Yaskawa INFORM job: DEMO_ROOF_SIDE_0625_3PAINT_22.JBI

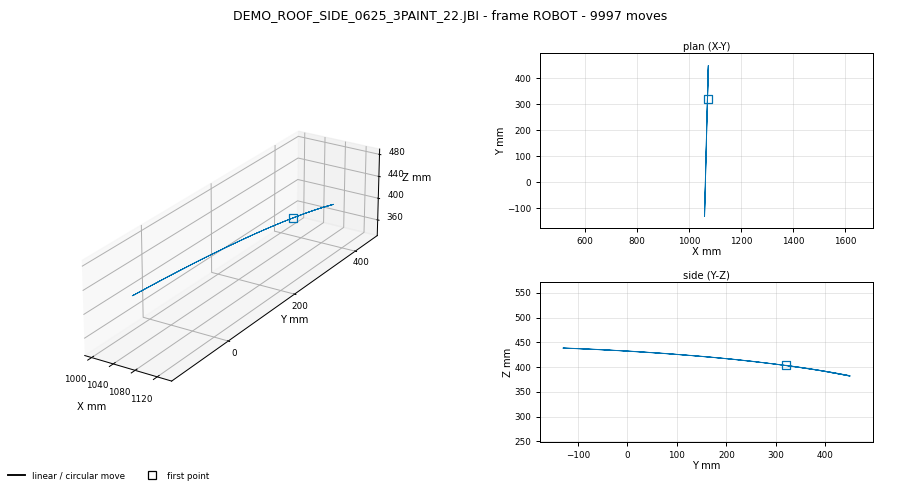
[picture p0: tool path of DEMO_ROOF_SIDE_0625_3PAINT_22.JBI in frame ROBOT, 9997 of 9997 moves have a stored position in this frame; points joined in program order, loops and branches not executed]
/JOB
//NAME DEMO_ROOF_SIDE_0625_3PAINT22
//POS
///NPOS 9997,0,0,0,0,0
///TOOL 0
///USER 0
///POSTYPE ROBOT
///RECTAN
///RCONF 1,0,0,0,0,0,0,0,0,0,0,0,0,0,0,0,0,0,0,0,0,0,0,0
C00000=1070.803,320.460,403.795,174.603,31.122,155.627
C00001=1070.809,320.707,403.762,174.607,31.127,155.628
C00002=1070.815,320.954,403.728,174.610,31.131,155.629
C00003=1070.822,321.203,403.695,174.613,31.136,155.630
C00004=1070.827,321.451,403.662,174.616,31.140,155.630
C00005=1070.834,321.698,403.629,174.620,31.145,155.631
C00006=1070.840,321.946,403.595,174.622,31.150,155.632
C00007=1070.846,322.193,403.562,174.626,31.155,155.633
C00008=1070.852,322.442,403.529,174.629,31.159,155.634
C00009=1070.859,322.689,403.495,174.633,31.164,155.635
C00010=1070.864,322.937,403.462,174.635,31.169,155.636
C00011=1070.870,323.184,403.429,174.639,31.173,155.636
C00012=1070.876,323.431,403.395,174.642,31.178,155.637
C00013=1070.883,323.680,403.362,174.645,31.183,155.638
C00014=1070.889,323.928,403.329,174.648,31.187,155.639
C00015=1070.895,324.175,403.295,174.652,31.192,155.640
C00016=1070.901,324.423,403.262,174.654,31.197,155.641
C00017=1070.908,324.670,403.228,174.658,31.201,155.642
C00018=1070.914,324.918,403.195,174.661,31.206,155.643
C00019=1070.920,325.165,403.161,174.665,31.211,155.643
C00020=1070.926,325.414,403.127,174.667,31.215,155.644
C00021=1070.933,325.661,403.094,174.671,31.220,155.645
C00022=1070.939,325.909,403.061,174.674,31.225,155.646
C00023=1070.946,326.156,403.027,174.677,31.230,155.647
C00024=1070.951,326.404,402.994,174.680,31.234,155.648
C00025=1070.957,326.651,402.959,174.684,31.239,155.649
C00026=1070.964,326.900,402.926,174.687,31.244,155.650
C00027=1070.970,327.147,402.892,174.690,31.249,155.650
C00028=1070.977,327.395,402.858,174.693,31.253,155.651
C00029=1070.983,327.643,402.825,174.697,31.258,155.652
C00030=1070.989,327.890,402.792,174.700,31.263,155.653
C00031=1070.996,328.138,402.757,174.703,31.268,155.654
C00032=1071.001,328.385,402.724,174.707,31.273,155.655
C00033=1071.008,328.633,402.690,174.710,31.277,155.656
C00034=1071.014,328.880,402.656,174.713,31.282,155.657
C00035=1071.022,329.128,402.622,174.716,31.287,155.658
C00036=1071.027,329.376,402.589,174.720,31.292,155.658
C00037=1071.034,329.624,402.554,174.722,31.296,155.659
C00038=1071.040,329.871,402.521,174.726,31.301,155.660
C00039=1071.047,330.119,402.487,174.730,31.306,155.661
C00040=1071.052,330.366,402.453,174.733,31.311,155.662
C00041=1071.058,330.589,402.423,174.735,31.315,155.663
C00042=1071.064,330.812,402.392,174.739,31.319,155.664
C00043=1071.070,331.035,402.362,174.742,31.324,155.664
C00044=1071.075,331.258,402.331,174.745,31.328,155.665
C00045=1071.081,331.480,402.300,174.747,31.332,155.666
C00046=1071.086,331.703,402.270,174.751,31.337,155.667
C00047=1071.092,331.926,402.239,174.754,31.341,155.668
C00048=1071.098,332.149,402.208,174.757,31.345,155.668
C00049=1071.104,332.397,402.174,174.760,31.350,155.669
C00050=1071.110,332.645,402.140,174.763,31.355,155.670
C00051=1071.116,332.892,402.105,174.767,31.360,155.671
C00052=1071.122,333.139,402.071,174.770,31.365,155.672
C00053=1071.129,333.387,402.036,174.773,31.370,155.673
C00054=1071.135,333.635,402.002,174.777,31.375,155.674
C00055=1071.141,333.882,401.968,174.780,31.380,155.675
C00056=1071.147,334.130,401.933,174.783,31.385,155.676
C00057=1071.153,334.377,401.899,174.787,31.390,155.677
C00058=1071.160,334.625,401.865,174.790,31.395,155.678
C00059=1071.166,334.872,401.831,174.794,31.400,155.679
C00060=1071.172,335.120,401.796,174.797,31.405,155.680
C00061=1071.178,335.367,401.762,174.800,31.410,155.681
C00062=1071.185,335.615,401.727,174.804,31.415,155.682
C00063=1071.191,335.863,401.693,174.806,31.420,155.683
C00064=1071.197,336.110,401.658,174.810,31.425,155.684
C00065=1071.204,336.358,401.624,174.814,31.430,155.684
C00066=1071.210,336.605,401.590,174.817,31.435,155.685
C00067=1071.216,336.853,401.555,174.820,31.440,155.686
C00068=1071.223,337.100,401.520,174.824,31.445,155.687
C00069=1071.229,337.348,401.486,174.827,31.450,155.688
C00070=1071.235,337.596,401.452,174.831,31.455,155.689
C00071=1071.242,337.843,401.416,174.834,31.460,155.690
C00072=1071.248,338.090,401.382,174.837,31.465,155.691
C00073=1071.255,338.338,401.347,174.841,31.470,155.692
C00074=1071.260,338.586,401.312,174.844,31.476,155.693
C00075=1071.266,338.833,401.277,174.847,31.480,155.694
C00076=1071.273,339.081,401.243,174.851,31.486,155.695
C00077=1071.280,339.328,401.208,174.855,31.491,155.696
C00078=1071.285,339.575,401.173,174.858,31.496,155.697
C00079=1071.292,339.823,401.138,174.861,31.501,155.698
C00080=1071.298,340.071,401.104,174.865,31.506,155.699
C00081=1071.304,340.317,401.069,174.869,31.511,155.700
C00082=1071.310,340.565,401.033,174.871,31.517,155.701
C00083=1071.317,340.813,400.999,174.875,31.522,155.702
C00084=1071.323,341.060,400.964,174.879,31.527,155.703
C00085=1071.329,341.307,400.928,174.883,31.532,155.704
C00086=1071.335,341.555,400.894,174.885,31.537,155.705
C00087=1071.342,341.803,400.859,174.889,31.543,155.706
C00088=1071.349,342.050,400.824,174.893,31.548,155.707
C00089=1071.354,342.298,400.789,174.896,31.553,155.708
C00090=1071.361,342.545,400.754,174.899,31.558,155.709
C00091=1071.368,342.793,400.719,174.903,31.563,155.710
C00092=1071.374,343.040,400.683,174.907,31.569,155.711
C00093=1071.380,343.288,400.649,174.910,31.573,155.712
C00094=1071.386,343.535,400.614,174.913,31.579,155.713
C00095=1071.392,343.783,400.578,174.917,31.584,155.714
C00096=1071.399,344.030,400.543,174.921,31.589,155.715
C00097=1071.405,344.250,400.511,174.924,31.594,155.716
C00098=1071.410,344.470,400.480,174.926,31.599,155.717
C00099=1071.416,344.691,400.449,174.930,31.604,155.718
C00100=1071.422,344.911,400.417,174.933,31.608,155.719
C00101=1071.426,345.131,400.386,174.936,31.613,155.719
C00102=1071.432,345.352,400.354,174.939,31.617,155.720
C00103=1071.438,345.572,400.323,174.942,31.622,155.721
C00104=1071.444,345.792,400.291,174.946,31.627,155.722
C00105=1071.450,346.039,400.256,174.949,31.632,155.723
C00106=1071.456,346.287,400.221,174.953,31.638,155.724
C00107=1071.462,346.535,400.185,174.956,31.643,155.725
C00108=1071.469,346.782,400.150,174.960,31.649,155.726
C00109=1071.475,347.029,400.113,174.963,31.654,155.727
C00110=1071.482,347.276,400.078,174.967,31.659,155.728
C00111=1071.488,347.524,400.042,174.970,31.665,155.729
C00112=1071.494,347.771,400.008,174.974,31.670,155.730
C00113=1071.500,348.018,399.972,174.978,31.676,155.732
C00114=1071.507,348.266,399.936,174.982,31.681,155.733
C00115=1071.514,348.513,399.900,174.984,31.686,155.734
C00116=1071.520,348.760,399.865,174.988,31.692,155.735
C00117=1071.526,349.008,399.829,174.992,31.697,155.736
C00118=1071.532,349.256,399.794,174.996,31.703,155.737
C00119=1071.539,349.503,399.757,174.999,31.708,155.738
C00120=1071.545,349.750,399.722,175.002,31.714,155.739
C00121=1071.552,349.998,399.686,175.006,31.719,155.740
C00122=1071.558,350.245,399.650,175.010,31.725,155.741
C00123=1071.564,350.492,399.614,175.013,31.730,155.742
C00124=1071.571,350.739,399.578,175.017,31.735,155.743
C00125=1071.577,350.987,399.543,175.021,31.741,155.744
C00126=1071.583,351.234,399.507,175.025,31.747,155.745
C00127=1071.590,351.481,399.471,175.028,31.752,155.746
C00128=1071.596,351.729,399.435,175.031,31.757,155.747
C00129=1071.602,351.976,399.399,175.035,31.763,155.749
C00130=1071.609,352.223,399.364,175.039,31.769,155.750
C00131=1071.616,352.471,399.327,175.043,31.774,155.751
C00132=1071.622,352.719,399.291,175.046,31.780,155.752
C00133=1071.629,352.966,399.255,175.050,31.785,155.753
C00134=1071.635,353.213,399.218,175.054,31.791,155.754
C00135=1071.641,353.460,399.183,175.057,31.797,155.755
C00136=1071.647,353.708,399.146,175.060,31.802,155.756
C00137=1071.654,353.954,399.110,175.064,31.808,155.757
C00138=1071.660,354.202,399.075,175.068,31.813,155.758
C00139=1071.667,354.449,399.038,175.072,31.819,155.760
C00140=1071.673,354.696,399.002,175.076,31.825,155.761
C00141=1071.679,354.944,398.966,175.079,31.831,155.762
C00142=1071.686,355.191,398.929,175.083,31.837,155.763
C00143=1071.692,355.439,398.893,175.087,31.842,155.764
C00144=1071.699,355.686,398.856,175.091,31.848,155.765
C00145=1071.705,355.933,398.820,175.094,31.854,155.766
C00146=1071.711,356.180,398.783,175.097,31.859,155.767
C00147=1071.717,356.427,398.748,175.101,31.865,155.769
C00148=1071.724,356.675,398.711,175.105,31.870,155.770
C00149=1071.731,356.922,398.674,175.109,31.876,155.771
C00150=1071.737,357.169,398.638,175.112,31.882,155.772
C00151=1071.743,357.416,398.601,175.116,31.888,155.773
C00152=1071.750,357.663,398.565,175.120,31.893,155.774
C00153=1071.756,357.886,398.532,175.124,31.899,155.775
C00154=1071.762,358.108,398.499,175.127,31.904,155.776
C00155=1071.767,358.330,398.466,175.130,31.909,155.777
C00156=1071.774,358.552,398.433,175.133,31.915,155.779
C00157=1071.780,358.774,398.401,175.137,31.919,155.779
C00158=1071.785,358.996,398.368,175.141,31.925,155.780
C00159=1071.791,359.218,398.335,175.144,31.930,155.782
C00160=1071.797,359.440,398.302,175.148,31.935,155.783
C00161=1071.803,359.688,398.265,175.151,31.941,155.784
C00162=1071.810,359.935,398.228,175.155,31.947,155.785
C00163=1071.816,360.182,398.192,175.159,31.953,155.786
C00164=1071.823,360.429,398.154,175.163,31.959,155.787
C00165=1071.830,360.676,398.118,175.167,31.965,155.788
C00166=1071.836,360.923,398.082,175.170,31.971,155.790
C00167=1071.842,361.170,398.045,175.174,31.977,155.791
C00168=1071.849,361.417,398.007,175.178,31.983,155.792
C00169=1071.855,361.665,397.971,175.182,31.988,155.793
C00170=1071.861,361.912,397.934,175.186,31.995,155.795
C00171=1071.869,362.159,397.897,175.189,32.001,155.796
C00172=1071.874,362.406,397.860,175.193,32.007,155.797
C00173=1071.881,362.654,397.823,175.197,32.012,155.798
C00174=1071.888,362.900,397.786,175.201,32.018,155.799
C00175=1071.894,363.147,397.749,175.205,32.025,155.801
C00176=1071.901,363.394,397.712,175.208,32.031,155.802
C00177=1071.907,363.642,397.675,175.212,32.037,155.803
C00178=1071.914,363.889,397.637,175.216,32.042,155.804
C00179=1071.921,364.136,397.601,175.220,32.049,155.805
C00180=1071.927,364.383,397.562,175.224,32.055,155.807
C00181=1071.933,364.631,397.526,175.228,32.061,155.808
C00182=1071.940,364.877,397.489,175.231,32.067,155.809
C00183=1071.947,365.124,397.451,175.235,32.073,155.810
C00184=1071.953,365.371,397.414,175.239,32.079,155.812
C00185=1071.959,365.619,397.376,175.243,32.086,155.813
C00186=1071.966,365.865,397.339,175.247,32.092,155.814
C00187=1071.972,366.113,397.302,175.250,32.098,155.815
C00188=1071.979,366.360,397.264,175.255,32.104,155.816
C00189=1071.985,366.607,397.226,175.259,32.110,155.818
C00190=1071.992,366.854,397.189,175.263,32.117,155.819
C00191=1071.998,367.102,397.152,175.267,32.123,155.820
C00192=1072.005,367.348,397.115,175.271,32.129,155.822
C00193=1072.011,367.596,397.076,175.274,32.135,155.823
C00194=1072.018,367.842,397.039,175.278,32.142,155.824
C00195=1072.025,368.090,397.001,175.282,32.148,155.825
C00196=1072.031,368.336,396.964,175.286,32.154,155.827
C00197=1072.038,368.583,396.926,175.290,32.160,155.828
C00198=1072.044,368.830,396.889,175.295,32.167,155.829
C00199=1072.051,369.077,396.851,175.298,32.173,155.831
C00200=1072.058,369.324,396.813,175.302,32.180,155.832
C00201=1072.064,369.571,396.775,175.306,32.186,155.833
C00202=1072.071,369.818,396.738,175.310,32.192,155.834
C00203=1072.077,370.065,396.700,175.314,32.198,155.836
C00204=1072.084,370.313,396.662,175.318,32.205,155.837
C00205=1072.090,370.559,396.625,175.322,32.211,155.838
C00206=1072.097,370.806,396.587,175.326,32.217,155.840
C00207=1072.104,371.054,396.549,175.330,32.224,155.841
C00208=1072.110,371.300,396.511,175.334,32.230,155.842
C00209=1072.117,371.531,396.476,175.338,32.237,155.844
C00210=1072.123,371.762,396.441,175.342,32.242,155.845
C00211=1072.129,371.992,396.405,175.346,32.248,155.846
C00212=1072.136,372.223,396.369,175.349,32.255,155.847
C00213=1072.141,372.453,396.334,175.353,32.260,155.848
C00214=1072.148,372.683,396.299,175.356,32.267,155.850
C00215=1072.155,372.914,396.263,175.360,32.272,155.851
C00216=1072.160,373.145,396.228,175.364,32.279,155.852
C00217=1072.167,373.392,396.189,175.369,32.285,155.854
C00218=1072.174,373.638,396.152,175.373,32.292,155.855
C00219=1072.181,373.885,396.113,175.377,32.299,155.856
C00220=1072.187,374.132,396.075,175.380,32.305,155.858
C00221=1072.193,374.378,396.036,175.384,32.312,155.859
C00222=1072.200,374.626,395.998,175.389,32.318,155.860
C00223=1072.207,374.873,395.959,175.393,32.325,155.862
C00224=1072.213,375.120,395.921,175.397,32.332,155.863
C00225=1072.219,375.366,395.883,175.401,32.338,155.865
C00226=1072.227,375.613,395.845,175.405,32.345,155.866
C00227=1072.233,375.860,395.806,175.410,32.352,155.867
C00228=1072.240,376.108,395.768,175.413,32.359,155.869
C00229=1072.247,376.355,395.729,175.417,32.365,155.870
C00230=1072.253,376.601,395.691,175.421,32.372,155.872
C00231=1072.259,376.848,395.653,175.426,32.379,155.873
C00232=1072.266,377.095,395.614,175.430,32.386,155.874
C00233=1072.273,377.342,395.575,175.434,32.392,155.876
C00234=1072.280,377.589,395.536,175.438,32.399,155.877
C00235=1072.286,377.836,395.498,175.443,32.406,155.879
C00236=1072.293,378.083,395.459,175.446,32.413,155.880
C00237=1072.299,378.329,395.421,175.450,32.420,155.881
C00238=1072.306,378.576,395.382,175.455,32.426,155.883
C00239=1072.313,378.823,395.343,175.459,32.433,155.884
C00240=1072.320,379.069,395.304,175.463,32.440,155.886
C00241=1072.327,379.316,395.266,175.468,32.447,155.887
C00242=1072.333,379.563,395.227,175.472,32.454,155.889
C00243=1072.340,379.810,395.188,175.476,32.461,155.890
C00244=1072.347,380.057,395.150,175.481,32.468,155.892
C00245=1072.354,380.304,395.110,175.485,32.475,155.893
C00246=1072.361,380.550,395.071,175.488,32.482,155.895
C00247=1072.367,380.797,395.032,175.493,32.489,155.896
C00248=1072.374,381.044,394.994,175.497,32.496,155.897
C00249=1072.381,381.291,394.955,175.501,32.503,155.899
C00250=1072.388,381.538,394.916,175.506,32.510,155.900
C00251=1072.395,381.784,394.877,175.510,32.517,155.902
C00252=1072.402,382.031,394.838,175.514,32.524,155.903
C00253=1072.408,382.278,394.799,175.519,32.531,155.905
C00254=1072.415,382.525,394.759,175.523,32.538,155.906
C00255=1072.422,382.771,394.720,175.527,32.545,155.908
C00256=1072.428,383.018,394.682,175.532,32.552,155.909
C00257=1072.435,383.264,394.642,175.536,32.560,155.911
C00258=1072.442,383.512,394.603,175.540,32.567,155.912
C00259=1072.448,383.758,394.564,175.544,32.574,155.914
C00260=1072.455,384.005,394.524,175.548,32.581,155.915
C00261=1072.462,384.252,394.485,175.553,32.589,155.917
C00262=1072.469,384.498,394.445,175.557,32.596,155.919
C00263=1072.476,384.746,394.406,175.561,32.603,155.920
C00264=1072.482,384.992,394.366,175.566,32.610,155.922
C00265=1072.490,385.237,394.327,175.570,32.618,155.923
C00266=1072.496,385.482,394.289,175.575,32.625,155.925
C00267=1072.502,385.727,394.249,175.579,32.633,155.926
C00268=1072.509,385.972,394.209,175.583,32.639,155.928
C00269=1072.516,386.217,394.171,175.588,32.647,155.929
C00270=1072.523,386.462,394.131,175.592,32.654,155.931
C00271=1072.530,386.709,394.091,175.597,32.662,155.933
C00272=1072.537,386.954,394.052,175.601,32.669,155.934
C00273=1072.544,387.200,394.013,175.606,32.676,155.936
C00274=1072.550,387.447,393.973,175.610,32.684,155.937
C00275=1072.557,387.693,393.933,175.615,32.692,155.939
C00276=1072.565,387.940,393.894,175.619,32.699,155.941
C00277=1072.571,388.187,393.854,175.624,32.706,155.942
C00278=1072.578,388.433,393.814,175.628,32.714,155.944
C00279=1072.585,388.680,393.774,175.632,32.722,155.945
C00280=1072.592,388.927,393.734,175.636,32.729,155.947
C00281=1072.599,389.173,393.694,175.641,32.736,155.948
C00282=1072.606,389.420,393.655,175.645,32.744,155.950
C00283=1072.613,389.667,393.615,175.650,32.752,155.952
C00284=1072.620,389.913,393.575,175.654,32.759,155.953
C00285=1072.627,390.160,393.535,175.659,32.767,155.955
C00286=1072.634,390.407,393.495,175.663,32.774,155.957
C00287=1072.641,390.653,393.455,175.668,32.782,155.958
C00288=1072.649,390.900,393.415,175.672,32.789,155.960
C00289=1072.655,391.146,393.375,175.677,32.797,155.962
C00290=1072.662,391.392,393.334,175.681,32.805,155.963
C00291=1072.669,391.639,393.294,175.686,32.813,155.965
C00292=1072.676,391.886,393.254,175.691,32.821,155.967
C00293=1072.683,392.133,393.214,175.695,32.828,155.968
C00294=1072.690,392.378,393.174,175.700,32.836,155.970
C00295=1072.697,392.625,393.133,175.704,32.844,155.972
C00296=1072.704,392.872,393.093,175.709,32.852,155.973
C00297=1072.711,393.118,393.053,175.713,32.860,155.975
C00298=1072.718,393.365,393.012,175.718,32.868,155.977
C00299=1072.724,393.612,392.972,175.723,32.876,155.979
C00300=1072.732,393.858,392.931,175.727,32.884,155.980
C00301=1072.739,394.104,392.891,175.732,32.892,155.982
C00302=1072.746,394.352,392.851,175.737,32.900,155.984
C00303=1072.752,394.597,392.810,175.742,32.908,155.985
C00304=1072.759,394.845,392.769,175.747,32.916,155.987
C00305=1072.766,395.091,392.728,175.751,32.924,155.989
C00306=1072.774,395.337,392.688,175.756,32.932,155.991
C00307=1072.781,395.584,392.647,175.761,32.940,155.993
C00308=1072.788,395.830,392.606,175.765,32.948,155.994
C00309=1072.795,396.077,392.566,175.770,32.956,155.996
C00310=1072.801,396.323,392.525,175.775,32.964,155.998
C00311=1072.808,396.570,392.485,175.779,32.972,156.000
C00312=1072.816,396.817,392.443,175.784,32.981,156.001
C00313=1072.822,397.063,392.402,175.789,32.989,156.003
C00314=1072.830,397.309,392.361,175.793,32.997,156.005
C00315=1072.837,397.556,392.321,175.798,33.005,156.007
C00316=1072.844,397.802,392.280,175.803,33.014,156.009
C00317=1072.851,398.049,392.239,175.807,33.022,156.010
C00318=1072.859,398.295,392.198,175.812,33.030,156.012
C00319=1072.866,398.542,392.157,175.817,33.038,156.014
C00320=1072.873,398.788,392.116,175.821,33.047,156.016
C00321=1072.879,399.048,392.072,175.827,33.056,156.018
C00322=1072.887,399.307,392.029,175.832,33.065,156.020
C00323=1072.894,399.567,391.986,175.837,33.073,156.022
C00324=1072.902,399.826,391.942,175.842,33.082,156.024
C00325=1072.909,400.072,391.902,175.847,33.091,156.026
C00326=1072.916,400.318,391.860,175.852,33.100,156.028
C00327=1072.923,400.565,391.819,175.857,33.108,156.029
C00328=1072.931,400.811,391.778,175.861,33.116,156.031
C00329=1072.938,401.058,391.735,175.866,33.125,156.033
C00330=1072.945,401.304,391.694,175.871,33.134,156.035
C00331=1072.952,401.550,391.653,175.877,33.142,156.037
C00332=1072.959,401.797,391.612,175.881,33.151,156.039
C00333=1072.966,402.043,391.571,175.886,33.160,156.041
C00334=1072.974,402.289,391.529,175.891,33.168,156.043
C00335=1072.981,402.536,391.488,175.896,33.177,156.045
C00336=1072.988,402.783,391.446,175.901,33.186,156.047
C00337=1072.995,403.029,391.404,175.906,33.195,156.049
C00338=1073.002,403.275,391.363,175.911,33.203,156.050
C00339=1073.010,403.522,391.321,175.916,33.212,156.052
C00340=1073.017,403.768,391.279,175.921,33.220,156.054
C00341=1073.024,404.015,391.238,175.926,33.229,156.056
C00342=1073.031,404.261,391.196,175.931,33.238,156.058
C00343=1073.038,404.508,391.154,175.936,33.247,156.060
C00344=1073.046,404.754,391.112,175.941,33.256,156.062
C00345=1073.053,405.000,391.070,175.946,33.265,156.064
C00346=1073.060,405.247,391.028,175.951,33.274,156.066
C00347=1073.067,405.492,390.986,175.956,33.283,156.068
C00348=1073.074,405.739,390.944,175.961,33.292,156.070
C00349=1073.082,405.985,390.902,175.966,33.301,156.072
C00350=1073.088,406.232,390.860,175.971,33.310,156.075
C00351=1073.096,406.478,390.818,175.977,33.319,156.077
C00352=1073.104,406.724,390.776,175.982,33.329,156.079
C00353=1073.111,406.971,390.734,175.987,33.337,156.081
C00354=1073.118,407.218,390.691,175.992,33.347,156.083
C00355=1073.125,407.463,390.649,175.997,33.356,156.085
C00356=1073.132,407.710,390.607,176.003,33.365,156.087
C00357=1073.140,407.956,390.565,176.008,33.374,156.089
C00358=1073.146,408.202,390.522,176.013,33.384,156.091
C00359=1073.154,408.449,390.479,176.018,33.393,156.093
C00360=1073.162,408.695,390.437,176.024,33.402,156.095
C00361=1073.168,408.941,390.395,176.029,33.412,156.097
C00362=1073.176,409.187,390.353,176.034,33.421,156.100
C00363=1073.183,409.434,390.310,176.039,33.431,156.102
C00364=1073.191,409.680,390.267,176.045,33.440,156.104
C00365=1073.198,409.926,390.225,176.050,33.449,156.106
C00366=1073.205,410.172,390.182,176.055,33.459,156.108
C00367=1073.212,410.419,390.139,176.060,33.469,156.110
C00368=1073.220,410.665,390.097,176.066,33.478,156.112
C00369=1073.227,410.911,390.054,176.071,33.488,156.115
C00370=1073.235,411.158,390.011,176.076,33.497,156.117
C00371=1073.242,411.404,389.969,176.081,33.507,156.119
C00372=1073.249,411.649,389.926,176.087,33.516,156.121
C00373=1073.257,411.896,389.883,176.092,33.526,156.123
C00374=1073.264,412.142,389.840,176.098,33.536,156.126
C00375=1073.272,412.388,389.798,176.103,33.546,156.128
C00376=1073.279,412.634,389.754,176.109,33.555,156.130
C00377=1073.287,412.898,389.709,176.114,33.566,156.132
C00378=1073.295,413.163,389.662,176.120,33.576,156.135
C00379=1073.304,413.427,389.617,176.127,33.587,156.137
C00380=1073.311,413.690,389.570,176.132,33.597,156.140
C00381=1073.319,413.936,389.527,176.137,33.607,156.142
C00382=1073.326,414.183,389.484,176.144,33.617,156.144
C00383=1073.334,414.429,389.441,176.149,33.627,156.146
C00384=1073.342,414.675,389.398,176.154,33.637,156.149
C00385=1073.350,414.921,389.354,176.160,33.647,156.151
C00386=1073.357,415.168,389.311,176.165,33.657,156.153
C00387=1073.364,415.413,389.268,176.171,33.667,156.156
C00388=1073.372,415.660,389.225,176.177,33.677,156.158
C00389=1073.379,415.905,389.181,176.182,33.687,156.160
C00390=1073.387,416.152,389.138,176.189,33.698,156.163
C00391=1073.395,416.398,389.094,176.194,33.707,156.165
C00392=1073.402,416.644,389.051,176.199,33.718,156.167
C00393=1073.410,416.890,389.007,176.205,33.728,156.170
C00394=1073.417,417.136,388.964,176.211,33.738,156.172
C00395=1073.424,417.382,388.920,176.216,33.748,156.174
C00396=1073.433,417.628,388.876,176.222,33.759,156.177
C00397=1073.439,417.874,388.832,176.228,33.770,156.179
C00398=1073.447,418.120,388.789,176.234,33.780,156.182
C00399=1073.454,418.367,388.745,176.239,33.790,156.184
C00400=1073.463,418.612,388.701,176.246,33.801,156.187
C00401=1073.470,418.858,388.657,176.251,33.811,156.189
C00402=1073.478,419.103,388.614,176.257,33.822,156.191
C00403=1073.485,419.348,388.570,176.263,33.832,156.194
C00404=1073.493,419.593,388.526,176.268,33.843,156.196
C00405=1073.501,419.839,388.482,176.275,33.853,156.199
C00406=1073.508,420.084,388.438,176.280,33.864,156.201
C00407=1073.516,420.329,388.394,176.287,33.874,156.204
C00408=1073.523,420.574,388.350,176.292,33.885,156.206
C00409=1073.531,420.820,388.306,176.299,33.896,156.209
C00410=1073.539,421.066,388.263,176.304,33.907,156.211
C00411=1073.547,421.312,388.218,176.311,33.918,156.214
C00412=1073.555,421.559,388.175,176.316,33.928,156.216
C00413=1073.562,421.805,388.130,176.323,33.939,156.219
C00414=1073.570,422.050,388.085,176.328,33.950,156.221
C00415=1073.577,422.296,388.040,176.335,33.961,156.224
C00416=1073.586,422.542,387.996,176.340,33.972,156.227
C00417=1073.594,422.788,387.952,176.347,33.983,156.229
C00418=1073.601,423.035,387.907,176.352,33.994,156.232
C00419=1073.608,423.280,387.863,176.359,34.005,156.234
C00420=1073.615,423.526,387.819,176.364,34.016,156.237
C00421=1073.623,423.771,387.774,176.371,34.028,156.240
C00422=1073.631,424.017,387.729,176.378,34.039,156.242
C00423=1073.639,424.263,387.684,176.383,34.050,156.245
C00424=1073.648,424.509,387.640,176.390,34.061,156.248
C00425=1073.655,424.755,387.595,176.395,34.073,156.250
C00426=1073.663,425.001,387.550,176.402,34.084,156.253
C00427=1073.671,425.247,387.505,176.408,34.095,156.256
C00428=1073.679,425.492,387.460,176.414,34.106,156.258
C00429=1073.686,425.738,387.415,176.421,34.118,156.261
C00430=1073.694,425.984,387.371,176.427,34.129,156.264
C00431=1073.702,426.229,387.325,176.434,34.141,156.266
C00432=1073.711,426.476,387.281,176.440,34.152,156.269
C00433=1073.719,426.757,387.229,176.447,34.166,156.272
C00434=1073.729,427.037,387.178,176.454,34.179,156.275
C00435=1073.737,427.318,387.126,176.462,34.192,156.278
C00436=1073.747,427.598,387.075,176.469,34.205,156.282
C00437=1073.755,427.844,387.029,176.475,34.217,156.284
C00438=1073.762,428.090,386.984,176.482,34.229,156.287
C00439=1073.770,428.336,386.938,176.489,34.241,156.290
C00440=1073.778,428.581,386.893,176.495,34.252,156.293
C00441=1073.786,428.828,386.848,176.501,34.264,156.296
C00442=1073.794,429.073,386.802,176.508,34.276,156.299
C00443=1073.802,429.318,386.757,176.515,34.288,156.301
C00444=1073.811,429.564,386.711,176.521,34.300,156.304
C00445=1073.818,429.810,386.666,176.528,34.313,156.307
C00446=1073.826,430.055,386.620,176.535,34.324,156.310
C00447=1073.835,430.301,386.575,176.542,34.336,156.313
C00448=1073.843,430.546,386.529,176.547,34.349,156.316
C00449=1073.850,430.792,386.483,176.554,34.361,156.319
C00450=1073.858,431.038,386.437,176.561,34.373,156.322
C00451=1073.866,431.283,386.392,176.568,34.385,156.325
C00452=1073.875,431.529,386.346,176.575,34.397,156.328
C00453=1073.883,431.774,386.300,176.581,34.410,156.331
C00454=1073.891,432.020,386.254,176.588,34.422,156.334
C00455=1073.899,432.266,386.208,176.595,34.435,156.337
C00456=1073.907,432.511,386.161,176.602,34.447,156.340
C00457=1073.915,432.757,386.116,176.609,34.460,156.343
C00458=1073.923,433.003,386.070,176.616,34.472,156.346
C00459=1073.931,433.248,386.023,176.623,34.485,156.349
C00460=1073.939,433.494,385.977,176.630,34.498,156.352
C00461=1073.947,433.738,385.931,176.636,34.510,156.355
C00462=1073.956,433.984,385.884,176.643,34.523,156.358
C00463=1073.964,434.230,385.838,176.650,34.536,156.361
C00464=1073.971,434.475,385.791,176.657,34.548,156.364
C00465=1073.980,434.721,385.745,176.665,34.561,156.368
C00466=1073.988,434.967,385.699,176.672,34.574,156.371
C00467=1073.996,435.212,385.652,176.679,34.587,156.374
C00468=1074.005,435.457,385.606,176.686,34.600,156.377
C00469=1074.013,435.703,385.559,176.693,34.613,156.380
C00470=1074.021,435.948,385.512,176.700,34.626,156.383
C00471=1074.030,436.193,385.466,176.707,34.639,156.387
C00472=1074.038,436.439,385.419,176.715,34.652,156.390
C00473=1074.047,436.684,385.372,176.722,34.665,156.393
C00474=1074.055,436.930,385.325,176.729,34.679,156.396
C00475=1074.063,437.175,385.279,176.736,34.692,156.399
C00476=1074.071,437.420,385.232,176.744,34.705,156.403
C00477=1074.080,437.666,385.185,176.751,34.718,156.406
C00478=1074.088,437.911,385.138,176.758,34.732,156.409
C00479=1074.097,438.156,385.091,176.765,34.745,156.413
C00480=1074.106,438.402,385.044,176.774,34.759,156.416
C00481=1074.114,438.647,384.996,176.781,34.772,156.419
C00482=1074.122,438.892,384.949,176.788,34.786,156.423
C00483=1074.131,439.138,384.903,176.796,34.799,156.426
C00484=1074.139,439.383,384.855,176.803,34.813,156.429
C00485=1074.147,439.629,384.808,176.810,34.827,156.433
C00486=1074.156,439.873,384.760,176.818,34.840,156.436
C00487=1074.164,440.119,384.712,176.826,34.854,156.440
C00488=1074.173,440.364,384.666,176.834,34.868,156.443
C00489=1074.186,440.768,384.587,176.846,34.891,156.449
C00490=1074.201,441.172,384.509,176.859,34.914,156.455
C00491=1074.215,441.576,384.431,176.871,34.937,156.460
C00492=1074.230,441.980,384.352,176.884,34.960,156.466
C00493=1074.238,442.225,384.304,176.892,34.975,156.470
C00494=1074.246,442.470,384.256,176.900,34.989,156.473
C00495=1074.255,442.715,384.208,176.908,35.003,156.477
C00496=1074.263,442.960,384.160,176.915,35.017,156.480
C00497=1074.272,443.205,384.112,176.924,35.032,156.484
C00498=1074.281,443.451,384.064,176.932,35.047,156.488
C00499=1074.289,443.696,384.016,176.939,35.061,156.491
C00500=1074.298,443.941,383.967,176.948,35.075,156.495
C00501=1074.307,444.186,383.920,176.955,35.090,156.499
C00502=1074.315,444.431,383.872,176.964,35.105,156.502
C00503=1074.324,444.676,383.823,176.972,35.119,156.506
C00504=1074.333,444.921,383.775,176.980,35.134,156.510
C00505=1074.342,445.166,383.726,176.988,35.149,156.514
C00506=1074.351,445.411,383.677,176.997,35.164,156.517
C00507=1074.359,445.656,383.629,177.005,35.179,156.521
C00508=1074.368,445.901,383.580,177.013,35.194,156.525
C00509=1074.377,446.146,383.532,177.021,35.209,156.529
C00510=1074.385,446.391,383.484,177.030,35.224,156.532
C00511=1074.394,446.636,383.435,177.038,35.239,156.536
C00512=1074.403,446.881,383.386,177.047,35.254,156.540
C00513=1074.412,447.126,383.338,177.054,35.269,156.544
C00514=1074.421,447.371,383.288,177.063,35.284,156.548
C00515=1074.430,447.616,383.240,177.071,35.300,156.552
C00516=1074.439,447.861,383.191,177.078,35.315,156.556
C00517=1074.448,448.105,383.142,177.085,35.330,156.560
C00518=1074.457,448.349,383.093,177.092,35.345,156.564
C00519=1074.466,448.593,383.045,177.098,35.360,156.567
C00520=1074.476,448.838,382.996,177.105,35.375,156.571
C00521=1074.487,449.082,382.948,177.111,35.389,156.575
C00522=1074.499,449.327,382.902,177.117,35.403,156.578
C00523=1074.514,449.573,382.856,177.123,35.416,156.582
C00524=1074.529,449.819,382.810,177.129,35.429,156.585
C00525=1074.173,449.816,382.569,177.111,35.579,156.625
C00526=1074.159,449.570,382.615,177.105,35.566,156.622
C00527=1074.145,449.325,382.661,177.099,35.553,156.618
C00528=1074.132,449.080,382.708,177.092,35.540,156.615
C00529=1074.120,448.835,382.755,177.087,35.526,156.611
C00530=1074.110,448.590,382.803,177.080,35.511,156.607
C00531=1074.101,448.346,382.853,177.073,35.496,156.603
C00532=1074.092,448.102,382.901,177.065,35.481,156.600
C00533=1074.083,447.858,382.950,177.059,35.466,156.596
C00534=1074.073,447.613,382.999,177.051,35.450,156.592
C00535=1074.065,447.369,383.048,177.043,35.435,156.588
C00536=1074.056,447.123,383.097,177.034,35.420,156.584
C00537=1074.047,446.878,383.146,177.027,35.405,156.580
C00538=1074.038,446.634,383.195,177.018,35.390,156.576
C00539=1074.029,446.389,383.243,177.009,35.375,156.572
C00540=1074.020,446.144,383.292,177.001,35.360,156.569
C00541=1074.011,445.899,383.341,176.992,35.345,156.565
C00542=1074.003,445.653,383.389,176.985,35.330,156.561
C00543=1073.993,445.409,383.438,176.976,35.315,156.557
C00544=1073.985,445.164,383.486,176.967,35.300,156.553
C00545=1073.976,444.919,383.536,176.959,35.285,156.550
C00546=1073.967,444.674,383.583,176.951,35.271,156.546
C00547=1073.959,444.429,383.632,176.943,35.256,156.542
C00548=1073.950,444.183,383.680,176.934,35.241,156.538
C00549=1073.941,443.939,383.728,176.927,35.227,156.535
C00550=1073.932,443.693,383.777,176.918,35.212,156.531
C00551=1073.924,443.448,383.825,176.910,35.198,156.527
C00552=1073.915,443.204,383.873,176.902,35.183,156.524
C00553=1073.907,442.958,383.921,176.894,35.169,156.520
C00554=1073.897,442.713,383.969,176.886,35.154,156.516
C00555=1073.889,442.468,384.017,176.878,35.140,156.513
C00556=1073.880,442.223,384.064,176.870,35.126,156.509
C00557=1073.872,441.978,384.112,176.862,35.112,156.506
C00558=1073.858,441.591,384.188,176.850,35.089,156.500
C00559=1073.845,441.206,384.263,176.837,35.067,156.495
C00560=1073.831,440.819,384.339,176.825,35.045,156.489
C00561=1073.817,440.433,384.413,176.813,35.023,156.484
C00562=1073.809,440.188,384.461,176.805,35.009,156.480
C00563=1073.801,439.943,384.508,176.797,34.996,156.477
C00564=1073.792,439.698,384.555,176.790,34.982,156.473
C00565=1073.784,439.453,384.603,176.783,34.968,156.470
C00566=1073.775,439.207,384.650,176.774,34.955,156.466
C00567=1073.767,438.962,384.698,176.767,34.941,156.463
C00568=1073.759,438.716,384.745,176.759,34.927,156.460
C00569=1073.750,438.472,384.792,176.752,34.914,156.456
C00570=1073.741,438.226,384.839,176.745,34.900,156.453
C00571=1073.732,437.981,384.886,176.737,34.887,156.450
C00572=1073.725,437.735,384.934,176.729,34.874,156.446
C00573=1073.716,437.490,384.980,176.722,34.860,156.443
C00574=1073.707,437.244,385.027,176.715,34.847,156.440
C00575=1073.699,436.999,385.075,176.707,34.834,156.437
C00576=1073.690,436.754,385.121,176.700,34.821,156.433
C00577=1073.682,436.508,385.168,176.693,34.808,156.430
C00578=1073.673,436.263,385.215,176.686,34.794,156.427
C00579=1073.666,436.018,385.262,176.678,34.781,156.424
C00580=1073.657,435.772,385.308,176.670,34.768,156.420
C00581=1073.649,435.527,385.355,176.663,34.755,156.417
C00582=1073.640,435.281,385.402,176.656,34.743,156.414
C00583=1073.632,435.036,385.448,176.649,34.729,156.411
C00584=1073.624,434.791,385.495,176.642,34.717,156.408
C00585=1073.615,434.545,385.541,176.635,34.704,156.405
C00586=1073.607,434.300,385.587,176.628,34.691,156.402
C00587=1073.599,434.054,385.634,176.621,34.678,156.398
C00588=1073.591,433.808,385.680,176.614,34.666,156.395
C00589=1073.583,433.563,385.726,176.606,34.653,156.392
C00590=1073.574,433.318,385.773,176.599,34.640,156.389
C00591=1073.567,433.073,385.819,176.592,34.628,156.386
C00592=1073.558,432.827,385.866,176.585,34.615,156.383
C00593=1073.550,432.581,385.912,176.578,34.602,156.380
C00594=1073.542,432.336,385.958,176.571,34.590,156.377
C00595=1073.534,432.090,386.004,176.564,34.578,156.374
C00596=1073.526,431.845,386.050,176.558,34.565,156.371
C00597=1073.517,431.599,386.096,176.552,34.553,156.368
C00598=1073.510,431.354,386.142,176.545,34.541,156.365
C00599=1073.502,431.107,386.188,176.538,34.529,156.362
C00600=1073.494,430.862,386.234,176.531,34.516,156.359
C00601=1073.485,430.617,386.280,176.524,34.504,156.356
C00602=1073.477,430.371,386.325,176.517,34.492,156.353
C00603=1073.469,430.126,386.371,176.510,34.480,156.350
C00604=1073.461,429.880,386.417,176.504,34.468,156.347
C00605=1073.453,429.634,386.463,176.497,34.455,156.344
C00606=1073.444,429.388,386.508,176.490,34.444,156.342
C00607=1073.437,429.143,386.554,176.484,34.432,156.339
C00608=1073.429,428.898,386.599,176.477,34.420,156.336
C00609=1073.421,428.651,386.645,176.471,34.408,156.333
C00610=1073.413,428.406,386.690,176.464,34.396,156.330
C00611=1073.405,428.160,386.735,176.457,34.384,156.327
C00612=1073.397,427.914,386.781,176.451,34.373,156.324
C00613=1073.389,427.669,386.826,176.444,34.361,156.322
C00614=1073.381,427.386,386.878,176.437,34.347,156.318
C00615=1073.371,427.104,386.930,176.429,34.334,156.315
C00616=1073.361,426.821,386.982,176.422,34.320,156.312
C00617=1073.352,426.539,387.033,176.414,34.307,156.309
C00618=1073.345,426.293,387.079,176.408,34.296,156.306
C00619=1073.337,426.048,387.123,176.402,34.284,156.303
C00620=1073.328,425.802,387.169,176.395,34.273,156.301
C00621=1073.320,425.556,387.214,176.388,34.262,156.298
C00622=1073.313,425.310,387.259,176.383,34.250,156.295
C00623=1073.305,425.065,387.304,176.376,34.239,156.292
C00624=1073.297,424.819,387.349,176.370,34.228,156.290
C00625=1073.289,424.573,387.393,176.364,34.216,156.287
C00626=1073.282,424.327,387.438,176.357,34.205,156.284
C00627=1073.273,424.082,387.483,176.351,34.194,156.282
C00628=1073.266,423.835,387.528,176.345,34.183,156.279
C00629=1073.257,423.589,387.573,176.338,34.171,156.277
C00630=1073.249,423.343,387.617,176.332,34.160,156.274
C00631=1073.242,423.097,387.662,176.326,34.149,156.271
C00632=1073.234,422.852,387.706,176.320,34.138,156.269
C00633=1073.227,422.606,387.751,176.314,34.127,156.266
C00634=1073.219,422.361,387.795,176.308,34.116,156.263
C00635=1073.211,422.115,387.839,176.301,34.105,156.261
C00636=1073.204,421.869,387.884,176.296,34.094,156.258
C00637=1073.196,421.622,387.928,176.289,34.083,156.256
C00638=1073.189,421.376,387.973,176.284,34.073,156.253
C00639=1073.181,421.131,388.017,176.277,34.062,156.251
C00640=1073.173,420.885,388.062,176.272,34.051,156.248
C00641=1073.165,420.639,388.105,176.265,34.040,156.246
C00642=1073.157,420.393,388.149,176.259,34.030,156.243
C00643=1073.149,420.146,388.193,176.253,34.019,156.241
C00644=1073.142,419.900,388.238,176.247,34.008,156.238
C00645=1073.134,419.655,388.281,176.241,33.998,156.236
C00646=1073.126,419.409,388.326,176.235,33.987,156.233
C00647=1073.119,419.163,388.369,176.230,33.977,156.231
C00648=1073.111,418.917,388.414,176.223,33.966,156.228
C00649=1073.103,418.670,388.457,176.218,33.956,156.226
C00650=1073.095,418.425,388.501,176.211,33.945,156.223
C00651=1073.088,418.179,388.545,176.206,33.935,156.221
C00652=1073.081,417.932,388.589,176.200,33.924,156.219
C00653=1073.073,417.686,388.633,176.194,33.914,156.216
C00654=1073.065,417.441,388.677,176.188,33.903,156.214
C00655=1073.058,417.195,388.720,176.183,33.893,156.211
C00656=1073.050,416.948,388.764,176.177,33.883,156.209
C00657=1073.043,416.703,388.807,176.171,33.872,156.207
C00658=1073.035,416.456,388.851,176.166,33.863,156.204
C00659=1073.027,416.210,388.894,176.159,33.852,156.202
C00660=1073.020,415.964,388.938,176.154,33.842,156.199
C00661=1073.012,415.718,388.981,176.148,33.832,156.197
C00662=1073.005,415.472,389.024,176.143,33.821,156.195
C00663=1072.997,415.226,389.068,176.136,33.812,156.192
C00664=1072.989,414.979,389.112,176.131,33.801,156.190
C00665=1072.982,414.734,389.155,176.126,33.792,156.188
C00666=1072.975,414.487,389.199,176.120,33.782,156.186
C00667=1072.967,414.242,389.241,176.115,33.772,156.183
C00668=1072.959,413.995,389.284,176.108,33.762,156.181
C00669=1072.951,413.749,389.328,176.103,33.752,156.179
C00670=1072.944,413.485,389.374,176.098,33.742,156.176
C00671=1072.936,413.221,389.420,176.091,33.731,156.174
C00672=1072.927,412.957,389.467,176.085,33.720,156.171
C00673=1072.919,412.692,389.512,176.080,33.710,156.169
C00674=1072.912,412.447,389.555,176.074,33.700,156.167
C00675=1072.905,412.200,389.598,176.069,33.690,156.165
C00676=1072.897,411.954,389.641,176.062,33.681,156.162
C00677=1072.889,411.708,389.683,176.057,33.671,156.160
C00678=1072.882,411.462,389.727,176.052,33.661,156.158
C00679=1072.875,411.215,389.770,176.046,33.652,156.156
C00680=1072.866,410.969,389.813,176.041,33.642,156.154
C00681=1072.859,410.723,389.855,176.036,33.633,156.151
C00682=1072.853,410.477,389.898,176.030,33.623,156.149
C00683=1072.844,410.231,389.941,176.025,33.614,156.147
C00684=1072.837,409.984,389.983,176.020,33.604,156.145
C00685=1072.830,409.738,390.026,176.015,33.595,156.143
C00686=1072.823,409.492,390.068,176.009,33.585,156.141
C00687=1072.815,409.245,390.111,176.004,33.576,156.139
C00688=1072.808,409.000,390.154,175.999,33.567,156.136
C00689=1072.801,408.754,390.196,175.993,33.557,156.134
C00690=1072.794,408.507,390.238,175.988,33.548,156.132
C00691=1072.786,408.260,390.281,175.983,33.539,156.130
C00692=1072.779,408.014,390.323,175.978,33.529,156.128
C00693=1072.772,407.768,390.366,175.972,33.520,156.126
C00694=1072.764,407.522,390.408,175.967,33.511,156.124
C00695=1072.757,407.276,390.450,175.962,33.501,156.122
C00696=1072.750,407.029,390.493,175.956,33.492,156.120
C00697=1072.742,406.783,390.535,175.951,33.483,156.118
C00698=1072.731,406.398,390.601,175.943,33.469,156.114
C00699=1072.720,406.012,390.666,175.934,33.455,156.111
C00700=1072.709,405.627,390.733,175.927,33.440,156.108
C00701=1072.697,405.241,390.799,175.919,33.427,156.105
C00702=1072.690,404.995,390.840,175.914,33.417,156.103
C00703=1072.683,404.748,390.882,175.908,33.408,156.101
C00704=1072.675,404.502,390.924,175.904,33.400,156.099
C00705=1072.669,404.255,390.966,175.899,33.391,156.097
C00706=1072.661,404.009,391.008,175.894,33.382,156.095
C00707=1072.654,403.763,391.049,175.888,33.373,156.093
C00708=1072.646,403.517,391.091,175.883,33.364,156.091
C00709=1072.640,403.270,391.133,175.878,33.355,156.089
C00710=1072.632,403.024,391.175,175.873,33.347,156.087
C00711=1072.625,402.777,391.216,175.869,33.338,156.085
C00712=1072.617,402.531,391.258,175.864,33.329,156.083
C00713=1072.611,402.284,391.300,175.858,33.321,156.081
C00714=1072.603,402.038,391.341,175.853,33.312,156.079
C00715=1072.596,401.791,391.382,175.848,33.303,156.077
C00716=1072.589,401.545,391.424,175.844,33.295,156.075
C00717=1072.581,401.299,391.466,175.839,33.286,156.073
C00718=1072.575,401.053,391.506,175.833,33.277,156.071
C00719=1072.568,400.806,391.548,175.828,33.269,156.070
C00720=1072.560,400.560,391.590,175.824,33.260,156.068
C00721=1072.553,400.313,391.631,175.819,33.252,156.066
C00722=1072.543,399.945,391.693,175.812,33.239,156.063
C00723=1072.532,399.577,391.755,175.805,33.226,156.060
C00724=1072.521,399.209,391.816,175.797,33.214,156.057
C00725=1072.511,398.841,391.878,175.790,33.201,156.055
C00726=1072.504,398.595,391.918,175.785,33.193,156.053
C00727=1072.497,398.348,391.960,175.780,33.185,156.051
C00728=1072.489,398.101,392.001,175.775,33.176,156.049
C00729=1072.482,397.855,392.042,175.771,33.168,156.047
C00730=1072.475,397.609,392.083,175.766,33.160,156.045
C00731=1072.468,397.362,392.124,175.760,33.152,156.044
C00732=1072.461,397.115,392.165,175.756,33.143,156.042
C00733=1072.454,396.869,392.206,175.751,33.135,156.040
C00734=1072.447,396.623,392.247,175.746,33.127,156.038
C00735=1072.439,396.376,392.287,175.742,33.119,156.036
C00736=1072.433,396.130,392.328,175.737,33.111,156.035
C00737=1072.425,395.883,392.369,175.732,33.103,156.033
C00738=1072.418,395.637,392.410,175.728,33.094,156.031
C00739=1072.412,395.390,392.450,175.723,33.086,156.029
C00740=1072.404,395.144,392.491,175.719,33.079,156.028
C00741=1072.398,394.897,392.532,175.713,33.070,156.026
C00742=1072.391,394.650,392.573,175.708,33.062,156.024
C00743=1072.384,394.404,392.612,175.704,33.054,156.022
C00744=1072.376,394.158,392.654,175.699,33.046,156.020
C00745=1072.369,393.910,392.694,175.695,33.038,156.019
C00746=1072.363,393.665,392.735,175.690,33.030,156.017
C00747=1072.355,393.418,392.775,175.685,33.022,156.015
C00748=1072.349,393.171,392.815,175.681,33.015,156.014
C00749=1072.341,392.925,392.856,175.676,33.007,156.012
C00750=1072.335,392.678,392.896,175.672,32.999,156.010
C00751=1072.327,392.431,392.936,175.667,32.991,156.009
C00752=1072.321,392.185,392.977,175.662,32.983,156.007
C00753=1072.314,391.939,393.017,175.658,32.975,156.005
C00754=1072.306,391.692,393.057,175.653,32.967,156.003
C00755=1072.300,391.445,393.097,175.649,32.960,156.002
C00756=1072.293,391.199,393.139,175.644,32.952,156.000
C00757=1072.286,390.953,393.178,175.640,32.944,155.998
C00758=1072.279,390.706,393.218,175.634,32.937,155.997
C00759=1072.272,390.459,393.258,175.630,32.929,155.995
C00760=1072.264,390.213,393.298,175.625,32.921,155.993
C00761=1072.257,389.966,393.338,175.621,32.913,155.992
C00762=1072.250,389.719,393.378,175.616,32.906,155.990
C00763=1072.244,389.473,393.418,175.612,32.899,155.989
C00764=1072.236,389.226,393.458,175.607,32.891,155.987
C00765=1072.230,388.980,393.498,175.602,32.883,155.985
C00766=1072.223,388.733,393.538,175.598,32.876,155.984
C00767=1072.215,388.486,393.578,175.593,32.868,155.982
C00768=1072.209,388.240,393.618,175.589,32.861,155.980
C00769=1072.202,387.994,393.657,175.585,32.854,155.979
C00770=1072.195,387.746,393.697,175.580,32.846,155.977
C00771=1072.188,387.500,393.737,175.576,32.838,155.976
C00772=1072.181,387.253,393.776,175.571,32.831,155.974
C00773=1072.174,387.007,393.816,175.567,32.824,155.972
C00774=1072.167,386.761,393.856,175.562,32.816,155.971
C00775=1072.160,386.515,393.895,175.558,32.809,155.969
C00776=1072.153,386.269,393.935,175.553,32.801,155.968
C00777=1072.146,386.023,393.974,175.549,32.794,155.966
C00778=1072.139,385.777,394.014,175.545,32.787,155.964
C00779=1072.133,385.531,394.053,175.540,32.779,155.963
C00780=1072.126,385.285,394.092,175.536,32.772,155.961
C00781=1072.119,385.040,394.132,175.531,32.765,155.960
C00782=1072.113,384.792,394.171,175.527,32.758,155.958
C00783=1072.106,384.546,394.211,175.523,32.750,155.957
C00784=1072.098,384.299,394.250,175.518,32.743,155.955
C00785=1072.092,384.052,394.290,175.514,32.736,155.954
C00786=1072.085,383.805,394.329,175.509,32.729,155.952
C00787=1072.078,383.559,394.368,175.505,32.721,155.951
C00788=1072.072,383.312,394.408,175.501,32.714,155.949
C00789=1072.065,383.065,394.447,175.496,32.707,155.948
C00790=1072.058,382.819,394.486,175.492,32.700,155.946
C00791=1072.051,382.572,394.525,175.488,32.692,155.944
C00792=1072.045,382.325,394.564,175.484,32.685,155.943
C00793=1072.038,382.079,394.604,175.480,32.678,155.941
C00794=1072.031,381.832,394.643,175.476,32.671,155.940
C00795=1072.025,381.585,394.682,175.471,32.664,155.938
C00796=1072.018,381.338,394.721,175.467,32.657,155.937
C00797=1072.012,381.091,394.760,175.462,32.650,155.935
C00798=1072.005,380.844,394.799,175.458,32.643,155.934
C00799=1071.998,380.598,394.838,175.454,32.636,155.932
C00800=1071.991,380.351,394.877,175.449,32.629,155.931
C00801=1071.984,380.105,394.916,175.445,32.622,155.930
C00802=1071.977,379.858,394.955,175.441,32.615,155.928
C00803=1071.970,379.611,394.994,175.437,32.608,155.927
C00804=1071.964,379.364,395.033,175.432,32.601,155.925
C00805=1071.957,379.117,395.071,175.428,32.595,155.924
C00806=1071.950,378.870,395.110,175.424,32.588,155.922
C00807=1071.943,378.623,395.148,175.419,32.581,155.921
C00808=1071.936,378.376,395.187,175.415,32.574,155.919
C00809=1071.929,378.130,395.225,175.411,32.567,155.918
C00810=1071.922,377.883,395.264,175.408,32.560,155.917
C00811=1071.916,377.636,395.303,175.403,32.553,155.915
C00812=1071.909,377.389,395.342,175.399,32.546,155.914
C00813=1071.903,377.142,395.380,175.395,32.540,155.912
C00814=1071.896,376.896,395.418,175.390,32.533,155.911
C00815=1071.889,376.649,395.457,175.386,32.526,155.910
C00816=1071.882,376.402,395.496,175.382,32.519,155.908
C00817=1071.876,376.154,395.534,175.378,32.513,155.907
C00818=1071.869,375.908,395.573,175.374,32.506,155.905
C00819=1071.862,375.661,395.612,175.369,32.499,155.904
C00820=1071.856,375.414,395.650,175.365,32.493,155.903
C00821=1071.850,375.167,395.689,175.361,32.486,155.901
C00822=1071.842,374.920,395.726,175.357,32.479,155.900
C00823=1071.835,374.673,395.765,175.353,32.473,155.898
C00824=1071.829,374.427,395.803,175.349,32.466,155.897
C00825=1071.823,374.180,395.842,175.345,32.460,155.896
C00826=1071.816,373.932,395.880,175.341,32.453,155.894
C00827=1071.809,373.685,395.918,175.337,32.446,155.893
C00828=1071.804,373.439,395.956,175.332,32.439,155.891
C00829=1071.797,373.192,395.995,175.328,32.433,155.890
C00830=1071.790,372.961,396.030,175.324,32.427,155.889
C00831=1071.784,372.730,396.067,175.320,32.421,155.888
C00832=1071.777,372.499,396.101,175.317,32.415,155.886
C00833=1071.771,372.267,396.137,175.314,32.409,155.885
C00834=1071.765,372.036,396.172,175.310,32.402,155.884
C00835=1071.759,371.805,396.208,175.306,32.397,155.883
C00836=1071.752,371.573,396.244,175.302,32.391,155.881
C00837=1071.746,371.342,396.279,175.298,32.384,155.880
C00838=1071.739,371.095,396.318,175.294,32.378,155.879
C00839=1071.733,370.849,396.355,175.290,32.372,155.877
C00840=1071.726,370.602,396.393,175.286,32.365,155.876
C00841=1071.719,370.354,396.431,175.281,32.359,155.875
C00842=1071.713,370.107,396.469,175.278,32.353,155.874
C00843=1071.706,369.860,396.506,175.274,32.346,155.872
C00844=1071.700,369.613,396.544,175.270,32.340,155.871
C00845=1071.693,369.366,396.581,175.266,32.333,155.870
C00846=1071.686,369.119,396.620,175.262,32.327,155.868
C00847=1071.680,368.873,396.657,175.258,32.321,155.867
C00848=1071.673,368.625,396.695,175.253,32.315,155.866
C00849=1071.666,368.378,396.732,175.249,32.308,155.864
C00850=1071.660,368.131,396.770,175.246,32.302,155.863
C00851=1071.654,367.884,396.808,175.242,32.296,155.862
C00852=1071.647,367.637,396.845,175.238,32.289,155.861
C00853=1071.640,367.390,396.884,175.234,32.283,155.859
C00854=1071.634,367.143,396.921,175.230,32.277,155.858
C00855=1071.627,366.896,396.959,175.226,32.271,155.857
C00856=1071.621,366.649,396.995,175.222,32.264,155.855
C00857=1071.614,366.401,397.033,175.218,32.258,155.854
C00858=1071.608,366.155,397.071,175.215,32.252,155.853
C00859=1071.601,365.908,397.109,175.211,32.246,155.852
C00860=1071.595,365.661,397.145,175.207,32.240,155.850
C00861=1071.588,365.413,397.183,175.202,32.233,155.849
C00862=1071.582,365.167,397.220,175.198,32.227,155.848
C00863=1071.576,364.920,397.258,175.194,32.221,155.847
C00864=1071.569,364.672,397.295,175.190,32.215,155.845
C00865=1071.562,364.426,397.332,175.187,32.209,155.844
C00866=1071.555,364.178,397.369,175.183,32.203,155.843
C00867=1071.550,363.931,397.407,175.179,32.197,155.842
C00868=1071.543,363.683,397.444,175.175,32.191,155.841
C00869=1071.536,363.437,397.481,175.171,32.185,155.839
C00870=1071.530,363.189,397.518,175.167,32.179,155.838
C00871=1071.523,362.943,397.555,175.164,32.172,155.837
C00872=1071.517,362.696,397.592,175.160,32.167,155.836
C00873=1071.510,362.448,397.629,175.156,32.161,155.834
C00874=1071.503,362.201,397.666,175.152,32.155,155.833
C00875=1071.497,361.954,397.704,175.148,32.148,155.832
C00876=1071.490,361.707,397.740,175.144,32.143,155.831
C00877=1071.484,361.460,397.777,175.140,32.137,155.830
C00878=1071.477,361.213,397.814,175.137,32.131,155.828
C00879=1071.470,360.966,397.851,175.133,32.125,155.827
C00880=1071.465,360.718,397.888,175.129,32.119,155.826
C00881=1071.458,360.470,397.925,175.125,32.113,155.825
C00882=1071.451,360.224,397.962,175.121,32.107,155.824
C00883=1071.445,359.977,397.998,175.117,32.101,155.823
C00884=1071.438,359.729,398.035,175.114,32.096,155.821
C00885=1071.432,359.482,398.071,175.110,32.090,155.820
C00886=1071.426,359.260,398.105,175.107,32.084,155.819
C00887=1071.420,359.037,398.138,175.103,32.079,155.818
C00888=1071.414,358.814,398.170,175.099,32.074,155.817
C00889=1071.408,358.591,398.204,175.096,32.068,155.816
C00890=1071.403,358.368,398.238,175.093,32.063,155.815
C00891=1071.397,358.146,398.270,175.090,32.058,155.814
C00892=1071.391,357.923,398.303,175.086,32.053,155.813
C00893=1071.385,357.700,398.335,175.083,32.048,155.812
C00894=1071.378,357.453,398.372,175.079,32.042,155.811
C00895=1071.372,357.205,398.408,175.075,32.036,155.809
C00896=1071.365,356.958,398.445,175.072,32.030,155.808
C00897=1071.359,356.711,398.481,175.068,32.025,155.807
C00898=1071.353,356.464,398.518,175.064,32.019,155.806
C00899=1071.346,356.217,398.555,175.060,32.013,155.805
C00900=1071.339,355.969,398.591,175.056,32.008,155.804
C00901=1071.333,355.722,398.628,175.052,32.002,155.803
C00902=1071.327,355.475,398.664,175.049,31.996,155.801
C00903=1071.320,355.228,398.700,175.045,31.990,155.800
C00904=1071.314,354.980,398.736,175.042,31.985,155.799
C00905=1071.307,354.733,398.773,175.038,31.979,155.798
C00906=1071.301,354.486,398.809,175.034,31.973,155.797
C00907=1071.295,354.239,398.846,175.031,31.967,155.796
C00908=1071.289,353.991,398.882,175.027,31.962,155.795
C00909=1071.282,353.744,398.918,175.023,31.956,155.794
C00910=1071.276,353.497,398.954,175.019,31.951,155.793
C00911=1071.269,353.250,398.990,175.015,31.945,155.791
C00912=1071.263,353.003,399.026,175.012,31.939,155.790
C00913=1071.256,352.755,399.063,175.009,31.934,155.789
C00914=1071.250,352.507,399.099,175.005,31.928,155.788
C00915=1071.244,352.260,399.135,175.001,31.923,155.787
C00916=1071.238,352.012,399.171,174.997,31.917,155.786
C00917=1071.230,351.766,399.207,174.994,31.912,155.785
C00918=1071.224,351.518,399.242,174.990,31.906,155.784
C00919=1071.218,351.271,399.279,174.986,31.900,155.783
C00920=1071.211,351.024,399.314,174.983,31.895,155.782
C00921=1071.205,350.777,399.350,174.979,31.890,155.781
C00922=1071.199,350.529,399.386,174.976,31.884,155.779
C00923=1071.192,350.282,399.422,174.972,31.879,155.778
C00924=1071.186,350.034,399.458,174.968,31.873,155.777
C00925=1071.180,349.787,399.493,174.964,31.867,155.776
C00926=1071.173,349.540,399.529,174.961,31.862,155.775
C00927=1071.167,349.292,399.565,174.958,31.857,155.774
C00928=1071.161,349.045,399.601,174.954,31.851,155.773
C00929=1071.154,348.798,399.637,174.950,31.846,155.772
C00930=1071.148,348.550,399.672,174.946,31.840,155.771
C00931=1071.142,348.303,399.708,174.943,31.835,155.770
C00932=1071.135,348.055,399.743,174.940,31.829,155.769
C00933=1071.128,347.808,399.780,174.936,31.824,155.768
C00934=1071.122,347.561,399.815,174.932,31.819,155.767
C00935=1071.116,347.313,399.850,174.928,31.813,155.766
C00936=1071.110,347.065,399.886,174.925,31.808,155.765
C00937=1071.103,346.818,399.921,174.922,31.803,155.763
C00938=1071.097,346.570,399.957,174.918,31.797,155.762
C00939=1071.090,346.324,399.993,174.914,31.792,155.761
C00940=1071.084,346.077,400.028,174.910,31.786,155.760
C00941=1071.078,345.829,400.063,174.908,31.781,155.759
C00942=1071.073,345.608,400.095,174.904,31.776,155.758
C00943=1071.066,345.387,400.127,174.901,31.772,155.758
C00944=1071.061,345.166,400.159,174.898,31.767,155.757
C00945=1071.055,344.945,400.190,174.894,31.762,155.756
C00946=1071.050,344.724,400.221,174.892,31.758,155.755
C00947=1071.044,344.504,400.253,174.889,31.753,155.754
C00948=1071.038,344.282,400.285,174.885,31.748,155.753
C00949=1071.033,344.061,400.316,174.882,31.743,155.752
C00950=1071.026,343.814,400.351,174.878,31.738,155.751
C00951=1071.020,343.566,400.387,174.875,31.733,155.750
C00952=1071.014,343.319,400.422,174.872,31.728,155.749
C00953=1071.007,343.072,400.457,174.868,31.722,155.748
C00954=1071.001,342.824,400.492,174.864,31.717,155.747
C00955=1070.995,342.576,400.527,174.860,31.712,155.746
C00956=1070.988,342.329,400.562,174.858,31.707,155.745
C00957=1070.981,342.081,400.598,174.854,31.702,155.744
C00958=1070.975,341.835,400.632,174.850,31.696,155.743
C00959=1070.970,341.587,400.667,174.847,31.691,155.742
C00960=1070.963,341.339,400.702,174.844,31.686,155.741
C00961=1070.956,341.092,400.738,174.840,31.681,155.740
C00962=1070.951,340.844,400.772,174.836,31.676,155.739
C00963=1070.944,340.597,400.807,174.833,31.670,155.738
C00964=1070.937,340.349,400.843,174.830,31.665,155.737
C00965=1070.931,340.101,400.877,174.826,31.660,155.736
C00966=1070.925,339.855,400.912,174.823,31.655,155.735
C00967=1070.919,339.607,400.947,174.819,31.650,155.734
C00968=1070.912,339.359,400.982,174.815,31.645,155.733
C00969=1070.906,339.113,401.017,174.813,31.640,155.732
C00970=1070.900,338.864,401.052,174.809,31.635,155.731
C00971=1070.894,338.617,401.087,174.805,31.629,155.730
C00972=1070.888,338.370,401.121,174.802,31.625,155.729
C00973=1070.881,338.122,401.156,174.799,31.619,155.728
C00974=1070.875,337.874,401.191,174.795,31.614,155.727
C00975=1070.869,337.627,401.225,174.792,31.609,155.726
C00976=1070.863,337.379,401.260,174.788,31.604,155.725
C00977=1070.856,337.131,401.295,174.785,31.599,155.724
C00978=1070.850,336.885,401.329,174.782,31.594,155.723
C00979=1070.843,336.637,401.364,174.778,31.589,155.722
C00980=1070.837,336.389,401.398,174.774,31.584,155.721
C00981=1070.831,336.142,401.433,174.772,31.579,155.721
C00982=1070.824,335.894,401.467,174.768,31.574,155.719
C00983=1070.819,335.647,401.501,174.764,31.569,155.719
C00984=1070.812,335.399,401.536,174.761,31.564,155.718
C00985=1070.805,335.151,401.571,174.758,31.559,155.717
C00986=1070.799,334.904,401.605,174.755,31.554,155.716
C00987=1070.793,334.656,401.639,174.751,31.549,155.715
C00988=1070.787,334.409,401.673,174.747,31.544,155.714
C00989=1070.781,334.161,401.708,174.745,31.539,155.713
C00990=1070.774,333.914,401.743,174.741,31.534,155.712
C00991=1070.768,333.666,401.777,174.738,31.529,155.711
C00992=1070.762,333.418,401.812,174.734,31.524,155.710
C00993=1070.756,333.171,401.846,174.731,31.519,155.709
C00994=1070.749,332.923,401.880,174.728,31.514,155.708
C00995=1070.743,332.676,401.914,174.724,31.509,155.707
C00996=1070.737,332.428,401.948,174.721,31.505,155.706
C00997=1070.731,332.180,401.983,174.718,31.500,155.705
C00998=1070.725,331.957,402.014,174.715,31.495,155.705
C00999=1070.720,331.734,402.044,174.712,31.491,155.704
C01000=1070.714,331.510,402.075,174.708,31.486,155.703
C01001=1070.709,331.286,402.106,174.705,31.482,155.702
C01002=1070.703,331.063,402.137,174.703,31.477,155.701
C01003=1070.697,330.840,402.167,174.700,31.473,155.700
C01004=1070.692,330.616,402.198,174.696,31.468,155.700
C01005=1070.685,330.392,402.228,174.693,31.464,155.699
C01006=1070.680,330.145,402.262,174.691,31.459,155.698
C01007=1070.673,329.897,402.297,174.687,31.454,155.697
C01008=1070.666,329.650,402.330,174.683,31.450,155.696
C01009=1070.660,329.402,402.365,174.680,31.445,155.695
C01010=1070.654,329.155,402.397,174.677,31.440,155.694
C01011=1070.647,328.907,402.432,174.674,31.436,155.693
C01012=1070.641,328.659,402.466,174.670,31.431,155.693
C01013=1070.634,328.412,402.500,174.667,31.426,155.692
C01014=1070.629,328.164,402.533,174.664,31.421,155.691
C01015=1070.621,327.916,402.567,174.661,31.417,155.690
C01016=1070.616,327.669,402.601,174.657,31.412,155.689
C01017=1070.610,327.422,402.635,174.654,31.407,155.688
C01018=1070.603,327.173,402.668,174.651,31.402,155.687
C01019=1070.597,326.926,402.702,174.647,31.397,155.686
C01020=1070.590,326.678,402.735,174.644,31.393,155.686
C01021=1070.584,326.430,402.769,174.640,31.388,155.685
C01022=1070.578,326.183,402.803,174.638,31.383,155.684
C01023=1070.571,325.935,402.836,174.634,31.379,155.683
C01024=1070.566,325.688,402.871,174.631,31.374,155.682
C01025=1070.559,325.440,402.903,174.628,31.369,155.681
C01026=1070.553,325.192,402.938,174.625,31.364,155.680
C01027=1070.547,324.944,402.970,174.621,31.360,155.679
C01028=1070.541,324.697,403.004,174.618,31.355,155.678
C01029=1070.534,324.449,403.038,174.615,31.350,155.678
C01030=1070.528,324.202,403.072,174.612,31.346,155.677
C01031=1070.522,323.954,403.104,174.608,31.341,155.676
C01032=1070.515,323.706,403.139,174.605,31.336,155.675
C01033=1070.509,323.458,403.172,174.602,31.332,155.674
C01034=1070.503,323.210,403.205,174.599,31.327,155.673
C01035=1070.497,322.963,403.238,174.595,31.323,155.672
C01036=1070.491,322.715,403.272,174.592,31.318,155.672
C01037=1070.484,322.467,403.305,174.590,31.313,155.671
C01038=1070.478,322.220,403.339,174.586,31.309,155.670
C01039=1070.472,321.972,403.372,174.583,31.304,155.669
C01040=1070.467,321.724,403.405,174.580,31.299,155.668
C01041=1070.459,321.477,403.439,174.577,31.294,155.667
C01042=1070.454,321.229,403.472,174.573,31.289,155.666
C01043=1070.448,320.981,403.505,174.570,31.285,155.665
C01044=1070.442,320.733,403.538,174.567,31.280,155.665
C01045=1070.435,320.486,403.572,174.564,31.276,155.664
C01046=1070.430,320.239,403.605,174.560,31.271,155.663
C01047=1070.423,319.990,403.638,174.557,31.267,155.662
C01048=1070.417,319.743,403.671,174.555,31.262,155.661
C01049=1070.411,319.495,403.704,174.551,31.257,155.660
C01050=1070.405,319.247,403.737,174.548,31.253,155.659
C01051=1070.399,319.000,403.771,174.545,31.248,155.659
C01052=1070.393,318.752,403.804,174.542,31.243,155.658
C01053=1070.387,318.504,403.837,174.539,31.239,155.657
C01054=1070.381,318.278,403.867,174.535,31.235,155.656
C01055=1070.376,318.052,403.897,174.533,31.230,155.655
C01056=1070.370,317.824,403.927,174.530,31.226,155.655
C01057=1070.364,317.598,403.957,174.527,31.222,155.654
C01058=1070.360,317.371,403.987,174.524,31.217,155.653
C01059=1070.353,317.145,404.018,174.522,31.213,155.652
C01060=1070.348,316.918,404.049,174.519,31.209,155.652
C01061=1070.343,316.692,404.078,174.516,31.205,155.651
C01062=1070.336,316.444,404.111,174.513,31.200,155.650
C01063=1070.331,316.196,404.144,174.510,31.196,155.649
C01064=1070.325,315.949,404.177,174.507,31.191,155.648
C01065=1070.319,315.701,404.209,174.503,31.187,155.647
C01066=1070.313,315.453,404.242,174.501,31.182,155.646
C01067=1070.307,315.205,404.275,174.497,31.177,155.646
C01068=1070.300,314.958,404.308,174.494,31.173,155.645
C01069=1070.295,314.710,404.341,174.492,31.168,155.644
C01070=1070.289,314.462,404.374,174.488,31.164,155.643
C01071=1070.282,314.214,404.407,174.485,31.159,155.642
C01072=1070.276,313.966,404.439,174.482,31.155,155.641
C01073=1070.270,313.719,404.472,174.479,31.150,155.641
C01074=1070.264,313.471,404.504,174.476,31.146,155.640
C01075=1070.258,313.223,404.536,174.472,31.141,155.639
C01076=1070.252,312.975,404.569,174.470,31.137,155.638
C01077=1070.245,312.728,404.602,174.467,31.133,155.637
C01078=1070.239,312.479,404.634,174.463,31.128,155.637
C01079=1070.233,312.232,404.667,174.460,31.124,155.636
C01080=1070.227,311.984,404.699,174.458,31.120,155.635
C01081=1070.220,311.736,404.731,174.454,31.115,155.634
C01082=1070.214,311.489,404.764,174.451,31.110,155.633
C01083=1070.208,311.241,404.796,174.448,31.106,155.633
C01084=1070.201,310.993,404.828,174.445,31.102,155.632
C01085=1070.195,310.745,404.861,174.442,31.097,155.631
C01086=1070.189,310.497,404.893,174.438,31.093,155.630
C01087=1070.183,310.250,404.926,174.436,31.089,155.629
C01088=1070.176,310.002,404.957,174.433,31.084,155.629
C01089=1070.170,309.754,404.990,174.429,31.080,155.628
C01090=1070.164,309.506,405.022,174.427,31.075,155.627
C01091=1070.157,309.258,405.055,174.424,31.071,155.626
C01092=1070.152,309.011,405.086,174.420,31.067,155.626
C01093=1070.146,308.763,405.118,174.417,31.062,155.625
C01094=1070.139,308.515,405.151,174.415,31.058,155.624
C01095=1070.133,308.267,405.183,174.411,31.054,155.623
C01096=1070.127,308.019,405.215,174.408,31.049,155.622
C01097=1070.121,307.771,405.247,174.406,31.045,155.622
C01098=1070.115,307.524,405.279,174.402,31.040,155.621
C01099=1070.109,307.276,405.312,174.399,31.036,155.620
C01100=1070.102,307.028,405.343,174.397,31.032,155.619
C01101=1070.096,306.780,405.375,174.393,31.027,155.618
C01102=1070.090,306.532,405.408,174.390,31.023,155.618
C01103=1070.085,306.285,405.440,174.387,31.019,155.617
C01104=1070.078,306.037,405.471,174.385,31.014,155.616
C01105=1070.072,305.789,405.503,174.381,31.010,155.615
C01106=1070.066,305.541,405.536,174.378,31.006,155.615
C01107=1070.060,305.293,405.568,174.376,31.001,155.614
C01108=1070.054,305.046,405.599,174.372,30.997,155.613
C01109=1070.048,304.798,405.631,174.369,30.992,155.612
C01110=1070.042,304.573,405.660,174.366,30.989,155.611
C01111=1070.037,304.348,405.690,174.364,30.984,155.611
C01112=1070.031,304.123,405.718,174.361,30.981,155.610
C01113=1070.026,303.898,405.747,174.358,30.977,155.609
C01114=1070.020,303.673,405.776,174.356,30.972,155.609
C01115=1070.015,303.449,405.805,174.353,30.969,155.608
C01116=1070.010,303.224,405.833,174.350,30.965,155.607
C01117=1070.004,302.999,405.862,174.347,30.961,155.606
C01118=1069.998,302.751,405.895,174.345,30.956,155.606
C01119=1069.992,302.504,405.926,174.342,30.952,155.605
C01120=1069.986,302.256,405.958,174.339,30.948,155.604
C01121=1069.980,302.008,405.990,174.336,30.944,155.603
C01122=1069.974,301.760,406.021,174.333,30.939,155.603
C01123=1069.967,301.512,406.053,174.330,30.935,155.602
C01124=1069.962,301.264,406.085,174.328,30.931,155.601
C01125=1069.956,301.017,406.117,174.324,30.926,155.600
C01126=1069.950,300.768,406.148,174.321,30.922,155.599
C01127=1069.944,300.521,406.179,174.319,30.918,155.599
C01128=1069.938,300.272,406.211,174.316,30.913,155.598
C01129=1069.933,300.025,406.243,174.312,30.909,155.597
C01130=1069.926,299.777,406.274,174.309,30.904,155.596
C01131=1069.920,299.529,406.306,174.307,30.900,155.596
C01132=1069.915,299.281,406.338,174.304,30.896,155.595
C01133=1069.908,299.033,406.369,174.301,30.891,155.594
C01134=1069.903,298.785,406.400,174.298,30.887,155.593
C01135=1069.897,298.537,406.432,174.295,30.883,155.593
C01136=1069.891,298.290,406.463,174.292,30.879,155.592
C01137=1069.885,298.042,406.495,174.290,30.874,155.591
C01138=1069.879,297.794,406.526,174.287,30.870,155.590
C01139=1069.873,297.546,406.558,174.283,30.866,155.589
C01140=1069.868,297.298,406.589,174.281,30.861,155.589
C01141=1069.861,297.050,406.621,174.278,30.857,155.588
C01142=1069.855,296.802,406.651,174.275,30.853,155.587
C01143=1069.849,296.554,406.683,174.273,30.849,155.586
C01144=1069.842,296.306,406.714,174.269,30.844,155.586
C01145=1069.837,296.058,406.745,174.266,30.840,155.585
C01146=1069.831,295.810,406.777,174.263,30.836,155.584
C01147=1069.825,295.562,406.807,174.261,30.832,155.583
C01148=1069.819,295.314,406.839,174.258,30.827,155.583
C01149=1069.813,295.067,406.870,174.254,30.823,155.582
C01150=1069.806,294.818,406.901,174.252,30.819,155.581
C01151=1069.801,294.571,406.933,174.249,30.815,155.580
C01152=1069.795,294.322,406.963,174.246,30.811,155.580
C01153=1069.788,294.075,406.994,174.244,30.807,155.579
C01154=1069.782,293.827,407.025,174.241,30.802,155.578
C01155=1069.777,293.578,407.056,174.237,30.798,155.577
C01156=1069.770,293.331,407.088,174.235,30.794,155.577
C01157=1069.764,293.083,407.118,174.232,30.790,155.576
C01158=1069.758,292.835,407.149,174.229,30.786,155.575
C01159=1069.753,292.587,407.180,174.227,30.781,155.574
C01160=1069.746,292.339,407.212,174.224,30.777,155.574
C01161=1069.740,292.091,407.242,174.220,30.773,155.573
C01162=1069.734,291.843,407.272,174.218,30.769,155.572
C01163=1069.728,291.595,407.304,174.215,30.764,155.571
C01164=1069.722,291.347,407.335,174.212,30.760,155.571
C01165=1069.716,291.099,407.366,174.210,30.756,155.570
C01166=1069.711,290.881,407.393,174.207,30.752,155.569
C01167=1069.706,290.664,407.419,174.204,30.749,155.569
C01168=1069.700,290.447,407.446,174.202,30.745,155.568
C01169=1069.695,290.229,407.473,174.200,30.742,155.567
C01170=1069.689,290.012,407.501,174.197,30.738,155.567
C01171=1069.684,289.794,407.528,174.194,30.734,155.566
C01172=1069.680,289.577,407.555,174.193,30.731,155.566
C01173=1069.674,289.360,407.581,174.190,30.727,155.565
C01174=1069.669,289.112,407.612,174.187,30.723,155.564
C01175=1069.662,288.864,407.643,174.184,30.719,155.563
C01176=1069.656,288.616,407.674,174.182,30.715,155.563
C01177=1069.650,288.367,407.704,174.178,30.711,155.562
C01178=1069.644,288.119,407.735,174.175,30.706,155.561
C01179=1069.638,287.872,407.765,174.173,30.702,155.561
C01180=1069.632,287.623,407.796,174.170,30.698,155.560
C01181=1069.626,287.375,407.826,174.167,30.694,155.559
C01182=1069.619,287.127,407.857,174.165,30.690,155.558
C01183=1069.614,286.879,407.887,174.162,30.685,155.558
C01184=1069.607,286.631,407.917,174.159,30.682,155.557
C01185=1069.601,286.383,407.948,174.157,30.677,155.556
C01186=1069.595,286.135,407.978,174.153,30.673,155.555
C01187=1069.589,285.887,408.008,174.150,30.669,155.555
C01188=1069.583,285.639,408.039,174.148,30.665,155.554
C01189=1069.577,285.391,408.070,174.145,30.661,155.553
C01190=1069.571,285.143,408.100,174.142,30.657,155.553
C01191=1069.565,284.895,408.130,174.140,30.653,155.552
C01192=1069.559,284.647,408.161,174.137,30.649,155.551
C01193=1069.553,284.399,408.191,174.134,30.644,155.550
C01194=1069.547,284.151,408.222,174.132,30.640,155.550
C01195=1069.541,283.903,408.252,174.129,30.636,155.549
C01196=1069.535,283.655,408.283,174.126,30.632,155.548
C01197=1069.529,283.406,408.312,174.124,30.628,155.547
C01198=1069.524,283.159,408.343,174.120,30.624,155.547
C01199=1069.517,282.911,408.372,174.117,30.620,155.546
C01200=1069.511,282.663,408.403,174.115,30.616,155.545
C01201=1069.505,282.415,408.434,174.112,30.611,155.545
C01202=1069.499,282.166,408.463,174.109,30.607,155.544
C01203=1069.493,281.918,408.493,174.107,30.603,155.543
C01204=1069.487,281.670,408.524,174.104,30.599,155.543
C01205=1069.481,281.422,408.555,174.102,30.595,155.542
C01206=1069.476,281.174,408.584,174.099,30.591,155.541
C01207=1069.470,280.926,408.615,174.096,30.587,155.540
C01208=1069.463,280.678,408.644,174.094,30.583,155.540
C01209=1069.458,280.430,408.674,174.091,30.578,155.539
C01210=1069.451,280.181,408.705,174.088,30.575,155.538
C01211=1069.446,279.934,408.735,174.086,30.571,155.538
C01212=1069.439,279.685,408.764,174.083,30.566,155.537
C01213=1069.433,279.438,408.794,174.080,30.563,155.536
C01214=1069.428,279.189,408.824,174.078,30.559,155.535
C01215=1069.421,278.941,408.854,174.075,30.554,155.535
C01216=1069.415,278.692,408.884,174.072,30.551,155.534
C01217=1069.409,278.445,408.914,174.070,30.546,155.533
C01218=1069.403,278.197,408.943,174.067,30.542,155.533
C01219=1069.397,277.949,408.974,174.064,30.538,155.532
C01220=1069.392,277.700,409.003,174.062,30.534,155.531
C01221=1069.385,277.453,409.033,174.059,30.530,155.530
C01222=1069.380,277.240,409.059,174.056,30.526,155.530
C01223=1069.375,277.028,409.084,174.054,30.523,155.529
C01224=1069.370,276.815,409.110,174.052,30.519,155.529
C01225=1069.365,276.603,409.135,174.049,30.516,155.528
C01226=1069.359,276.391,409.161,174.047,30.512,155.527
C01227=1069.355,276.179,409.186,174.045,30.509,155.527
C01228=1069.349,275.966,409.211,174.043,30.506,155.526
C01229=1069.344,275.755,409.237,174.040,30.502,155.526
C01230=1069.339,275.506,409.266,174.038,30.498,155.525
C01231=1069.333,275.257,409.296,174.035,30.494,155.524
C01232=1069.326,275.010,409.326,174.032,30.490,155.524
C01233=1069.320,274.761,409.356,174.030,30.486,155.523
C01234=1069.314,274.513,409.385,174.027,30.482,155.522
C01235=1069.308,274.265,409.415,174.024,30.478,155.521
C01236=1069.302,274.017,409.444,174.022,30.474,155.521
C01237=1069.297,273.769,409.474,174.019,30.470,155.520
C01238=1069.290,273.520,409.503,174.016,30.466,155.519
C01239=1069.285,273.273,409.533,174.014,30.462,155.519
C01240=1069.279,273.024,409.563,174.011,30.458,155.518
C01241=1069.273,272.776,409.592,174.009,30.454,155.517
C01242=1069.267,272.528,409.621,174.006,30.449,155.516
C01243=1069.261,272.280,409.651,174.003,30.446,155.516
C01244=1069.255,272.032,409.680,174.001,30.442,155.515
C01245=1069.249,271.784,409.710,173.998,30.437,155.514
C01246=1069.243,271.535,409.739,173.995,30.433,155.514
C01247=1069.237,271.287,409.768,173.993,30.430,155.513
C01248=1069.231,271.039,409.798,173.990,30.425,155.512
C01249=1069.225,270.791,409.827,173.988,30.422,155.512
C01250=1069.219,270.542,409.856,173.986,30.418,155.511
C01251=1069.213,270.294,409.885,173.983,30.414,155.510
C01252=1069.207,270.046,409.914,173.980,30.409,155.509
C01253=1069.201,269.798,409.944,173.978,30.406,155.509
C01254=1069.195,269.549,409.973,173.975,30.402,155.508
C01255=1069.189,269.301,410.003,173.973,30.397,155.507
C01256=1069.183,269.053,410.032,173.970,30.393,155.507
C01257=1069.177,268.805,410.061,173.967,30.390,155.506
C01258=1069.171,268.557,410.090,173.965,30.385,155.505
C01259=1069.165,268.308,410.120,173.962,30.381,155.505
C01260=1069.159,268.060,410.149,173.959,30.377,155.504
C01261=1069.153,267.812,410.178,173.957,30.374,155.503
C01262=1069.146,267.564,410.207,173.954,30.369,155.503
C01263=1069.141,267.315,410.236,173.951,30.365,155.502
C01264=1069.135,267.067,410.265,173.949,30.361,155.501
C01265=1069.129,266.820,410.294,173.947,30.358,155.501
C01266=1069.123,266.571,410.322,173.944,30.353,155.500
C01267=1069.118,266.323,410.352,173.942,30.349,155.499
C01268=1069.111,266.074,410.381,173.939,30.346,155.499
C01269=1069.105,265.826,410.410,173.937,30.341,155.498
C01270=1069.099,265.578,410.439,173.934,30.337,155.497
C01271=1069.093,265.329,410.467,173.931,30.333,155.496
C01272=1069.087,265.081,410.497,173.929,30.330,155.496
C01273=1069.081,264.833,410.526,173.926,30.325,155.495
C01274=1069.075,264.585,410.555,173.923,30.321,155.494
C01275=1069.070,264.337,410.583,173.921,30.317,155.494
C01276=1069.064,264.088,410.613,173.919,30.313,155.493
C01277=1069.058,263.840,410.642,173.916,30.309,155.492
C01278=1069.052,263.630,410.666,173.914,30.306,155.492
C01279=1069.047,263.419,410.691,173.912,30.303,155.491
C01280=1069.042,263.209,410.715,173.909,30.299,155.491
C01281=1069.037,262.998,410.738,173.908,30.296,155.490
C01282=1069.032,262.788,410.763,173.905,30.293,155.489
C01283=1069.027,262.577,410.788,173.903,30.289,155.489
C01284=1069.022,262.366,410.812,173.901,30.286,155.488
C01285=1069.016,262.156,410.836,173.899,30.282,155.488
C01286=1069.010,261.907,410.865,173.896,30.279,155.487
C01287=1069.004,261.659,410.894,173.894,30.275,155.486
C01288=1068.998,261.410,410.921,173.891,30.271,155.486
C01289=1068.991,261.162,410.951,173.888,30.267,155.485
C01290=1068.986,260.914,410.978,173.887,30.263,155.484
C01291=1068.980,260.666,411.007,173.884,30.259,155.484
C01292=1068.974,260.417,411.036,173.882,30.255,155.483
C01293=1068.968,260.169,411.065,173.879,30.251,155.482
C01294=1068.962,259.920,411.093,173.876,30.247,155.482
C01295=1068.955,259.672,411.122,173.874,30.243,155.481
C01296=1068.949,259.425,411.150,173.871,30.239,155.480
C01297=1068.943,259.176,411.179,173.868,30.235,155.480
C01298=1068.937,258.928,411.207,173.867,30.231,155.479
C01299=1068.931,258.679,411.235,173.864,30.227,155.478
C01300=1068.925,258.431,411.264,173.862,30.223,155.478
C01301=1068.920,258.183,411.292,173.859,30.220,155.477
C01302=1068.913,257.934,411.320,173.856,30.216,155.476
C01303=1068.907,257.686,411.349,173.854,30.212,155.476
C01304=1068.901,257.438,411.377,173.851,30.207,155.475
C01305=1068.895,257.189,411.405,173.849,30.204,155.474
C01306=1068.889,256.941,411.434,173.847,30.200,155.474
C01307=1068.883,256.692,411.463,173.844,30.196,155.473
C01308=1068.877,256.445,411.490,173.842,30.192,155.472
C01309=1068.871,256.197,411.519,173.839,30.188,155.472
C01310=1068.865,255.948,411.547,173.836,30.184,155.471
C01311=1068.859,255.699,411.576,173.835,30.180,155.470
C01312=1068.854,255.451,411.604,173.832,30.176,155.469
C01313=1068.847,255.203,411.631,173.829,30.172,155.469
C01314=1068.841,254.954,411.660,173.827,30.168,155.468
C01315=1068.835,254.706,411.688,173.824,30.164,155.467
C01316=1068.829,254.458,411.717,173.822,30.160,155.467
C01317=1068.823,254.209,411.745,173.820,30.156,155.466
C01318=1068.817,253.961,411.772,173.817,30.152,155.465
C01319=1068.811,253.712,411.801,173.815,30.148,155.465
C01320=1068.806,253.464,411.829,173.812,30.144,155.464
C01321=1068.800,253.216,411.858,173.810,30.140,155.463
C01322=1068.793,252.968,411.886,173.808,30.136,155.463
C01323=1068.788,252.720,411.913,173.805,30.132,155.462
C01324=1068.782,252.471,411.942,173.803,30.128,155.461
C01325=1068.776,252.222,411.970,173.800,30.124,155.461
C01326=1068.771,251.974,411.998,173.797,30.120,155.460
C01327=1068.764,251.726,412.026,173.796,30.116,155.459
C01328=1068.758,251.478,412.054,173.793,30.112,155.459
C01329=1068.753,251.229,412.082,173.791,30.108,155.458
C01330=1068.746,250.981,412.109,173.788,30.104,155.457
C01331=1068.741,250.732,412.138,173.785,30.100,155.456
C01332=1068.735,250.484,412.166,173.784,30.096,155.456
C01333=1068.729,250.236,412.194,173.781,30.092,155.455
C01334=1068.724,250.025,412.218,173.780,30.089,155.454
C01335=1068.719,249.812,412.241,173.777,30.085,155.454
C01336=1068.714,249.601,412.265,173.775,30.082,155.453
C01337=1068.709,249.389,412.289,173.773,30.078,155.453
C01338=1068.704,249.177,412.312,173.771,30.075,155.452
C01339=1068.700,248.965,412.337,173.769,30.072,155.452
C01340=1068.694,248.754,412.361,173.767,30.068,155.451
C01341=1068.689,248.542,412.384,173.765,30.065,155.450
C01342=1068.683,248.293,412.412,173.762,30.061,155.450
C01343=1068.678,248.045,412.440,173.761,30.057,155.449
C01344=1068.671,247.797,412.468,173.758,30.053,155.448
C01345=1068.666,247.549,412.496,173.756,30.049,155.448
C01346=1068.660,247.299,412.523,173.753,30.044,155.447
C01347=1068.654,247.051,412.550,173.751,30.041,155.446
C01348=1068.648,246.803,412.579,173.749,30.037,155.446
C01349=1068.643,246.555,412.607,173.746,30.032,155.445
C01350=1068.637,246.306,412.634,173.744,30.028,155.444
C01351=1068.631,246.058,412.662,173.742,30.025,155.444
C01352=1068.625,245.810,412.689,173.739,30.021,155.443
C01353=1068.620,245.560,412.717,173.737,30.017,155.442
C01354=1068.613,245.313,412.744,173.734,30.012,155.441
C01355=1068.608,245.064,412.772,173.733,30.009,155.441
C01356=1068.602,244.816,412.799,173.730,30.005,155.440
C01357=1068.595,244.567,412.827,173.727,30.001,155.440
C01358=1068.590,244.319,412.855,173.725,29.996,155.439
C01359=1068.583,244.070,412.882,173.723,29.993,155.438
C01360=1068.578,243.822,412.910,173.721,29.989,155.437
C01361=1068.572,243.573,412.937,173.718,29.985,155.437
C01362=1068.566,243.325,412.965,173.715,29.980,155.436
C01363=1068.560,243.077,412.992,173.714,29.977,155.435
C01364=1068.555,242.828,413.020,173.711,29.973,155.435
C01365=1068.549,242.580,413.047,173.709,29.969,155.434
C01366=1068.542,242.331,413.074,173.707,29.965,155.433
C01367=1068.537,242.083,413.102,173.704,29.961,155.433
C01368=1068.530,241.834,413.129,173.702,29.957,155.432
C01369=1068.524,241.586,413.156,173.699,29.953,155.431
C01370=1068.519,241.338,413.183,173.698,29.949,155.431
C01371=1068.513,241.088,413.211,173.695,29.945,155.430
C01372=1068.507,240.841,413.238,173.692,29.941,155.429
C01373=1068.500,240.592,413.265,173.691,29.937,155.429
C01374=1068.494,240.344,413.292,173.688,29.933,155.428
C01375=1068.489,240.095,413.320,173.686,29.929,155.427
C01376=1068.483,239.846,413.347,173.683,29.925,155.427
C01377=1068.477,239.598,413.374,173.681,29.922,155.426
C01378=1068.471,239.349,413.401,173.679,29.917,155.425
C01379=1068.465,239.101,413.428,173.676,29.913,155.425
C01380=1068.459,238.853,413.456,173.675,29.909,155.424
C01381=1068.453,238.604,413.483,173.672,29.906,155.423
C01382=1068.447,238.355,413.509,173.670,29.902,155.423
C01383=1068.441,238.108,413.537,173.668,29.898,155.422
C01384=1068.435,237.859,413.564,173.665,29.893,155.421
C01385=1068.429,237.610,413.590,173.663,29.889,155.421
C01386=1068.424,237.362,413.618,173.661,29.886,155.420
C01387=1068.417,237.113,413.645,173.659,29.882,155.419
C01388=1068.412,236.865,413.672,173.656,29.878,155.419
C01389=1068.406,236.616,413.699,173.654,29.874,155.418
C01390=1068.400,236.402,413.723,173.652,29.870,155.417
C01391=1068.395,236.186,413.746,173.650,29.867,155.417
C01392=1068.390,235.971,413.769,173.649,29.863,155.416
C01393=1068.385,235.756,413.793,173.646,29.860,155.416
C01394=1068.380,235.542,413.815,173.644,29.856,155.415
C01395=1068.375,235.326,413.839,173.643,29.853,155.414
C01396=1068.370,235.112,413.862,173.640,29.850,155.414
C01397=1068.365,234.897,413.885,173.638,29.846,155.413
C01398=1068.359,234.648,413.912,173.636,29.842,155.412
C01399=1068.353,234.399,413.939,173.634,29.838,155.412
C01400=1068.347,234.151,413.966,173.632,29.834,155.411
C01401=1068.341,233.902,413.992,173.630,29.830,155.410
C01402=1068.335,233.655,414.020,173.628,29.826,155.410
C01403=1068.329,233.406,414.046,173.625,29.822,155.409
C01404=1068.323,233.157,414.073,173.623,29.818,155.408
C01405=1068.317,232.909,414.100,173.621,29.814,155.408
C01406=1068.312,232.661,414.127,173.618,29.810,155.407
C01407=1068.306,232.412,414.153,173.617,29.806,155.406
C01408=1068.299,232.163,414.180,173.614,29.802,155.406
C01409=1068.294,231.915,414.207,173.612,29.798,155.405
C01410=1068.288,231.666,414.234,173.610,29.794,155.404
C01411=1068.282,231.417,414.260,173.607,29.790,155.404
C01412=1068.277,231.169,414.286,173.605,29.786,155.403
C01413=1068.270,230.920,414.313,173.603,29.782,155.402
C01414=1068.264,230.672,414.340,173.601,29.778,155.402
C01415=1068.259,230.423,414.367,173.599,29.774,155.401
C01416=1068.253,230.175,414.393,173.597,29.770,155.400
C01417=1068.247,229.927,414.420,173.594,29.766,155.400
C01418=1068.241,229.678,414.447,173.592,29.762,155.399
C01419=1068.234,229.430,414.473,173.590,29.758,155.398
C01420=1068.229,229.181,414.499,173.587,29.754,155.398
C01421=1068.223,228.932,414.525,173.586,29.750,155.397
C01422=1068.217,228.684,414.552,173.583,29.746,155.396
C01423=1068.211,228.435,414.579,173.582,29.742,155.395
C01424=1068.204,228.187,414.605,173.579,29.738,155.395
C01425=1068.199,227.938,414.631,173.576,29.734,155.394
C01426=1068.193,227.689,414.658,173.575,29.730,155.393
C01427=1068.187,227.441,414.684,173.572,29.726,155.393
C01428=1068.181,227.193,414.710,173.571,29.722,155.392
C01429=1068.175,226.943,414.737,173.568,29.718,155.391
C01430=1068.169,226.695,414.763,173.566,29.714,155.391
C01431=1068.163,226.447,414.790,173.564,29.710,155.390
C01432=1068.157,226.198,414.815,173.562,29.706,155.389
C01433=1068.151,225.950,414.842,173.560,29.702,155.389
C01434=1068.145,225.701,414.869,173.557,29.699,155.388
C01435=1068.140,225.452,414.895,173.555,29.694,155.387
C01436=1068.133,225.204,414.921,173.553,29.690,155.387
C01437=1068.128,224.955,414.947,173.551,29.686,155.386
C01438=1068.122,224.707,414.973,173.549,29.683,155.385
C01439=1068.115,224.458,415.000,173.547,29.678,155.385
C01440=1068.110,224.209,415.026,173.545,29.674,155.384
C01441=1068.104,223.961,415.052,173.543,29.670,155.383
C01442=1068.098,223.712,415.078,173.540,29.666,155.383
C01443=1068.092,223.464,415.104,173.538,29.662,155.382
C01444=1068.086,223.215,415.131,173.536,29.658,155.381
C01445=1068.081,222.966,415.157,173.534,29.654,155.381
C01446=1068.076,222.748,415.180,173.532,29.650,155.380
C01447=1068.070,222.528,415.203,173.530,29.647,155.379
C01448=1068.065,222.310,415.226,173.529,29.643,155.379
C01449=1068.060,222.091,415.249,173.527,29.640,155.378
C01450=1068.055,221.871,415.272,173.524,29.636,155.378
C01451=1068.050,221.653,415.295,173.523,29.633,155.377
C01452=1068.044,221.433,415.318,173.521,29.629,155.376
C01453=1068.039,221.215,415.341,173.520,29.626,155.376
C01454=1068.033,220.966,415.366,173.517,29.622,155.375
C01455=1068.027,220.717,415.393,173.515,29.618,155.374
C01456=1068.021,220.469,415.418,173.513,29.613,155.374
C01457=1068.015,220.220,415.443,173.510,29.609,155.373
C01458=1068.009,219.972,415.470,173.509,29.606,155.372
C01459=1068.003,219.723,415.495,173.506,29.602,155.372
C01460=1067.998,219.474,415.521,173.505,29.598,155.371
C01461=1067.991,219.226,415.547,173.502,29.593,155.370
C01462=1067.986,218.977,415.573,173.501,29.590,155.370
C01463=1067.979,218.728,415.599,173.498,29.586,155.369
C01464=1067.974,218.480,415.625,173.496,29.582,155.368
C01465=1067.967,218.231,415.651,173.494,29.577,155.367
C01466=1067.962,217.982,415.677,173.492,29.574,155.367
C01467=1067.955,217.734,415.703,173.490,29.570,155.366
C01468=1067.949,217.486,415.728,173.487,29.565,155.365
C01469=1067.944,217.237,415.754,173.486,29.561,155.365
C01470=1067.938,216.988,415.779,173.483,29.557,155.364
C01471=1067.932,216.739,415.805,173.482,29.553,155.363
C01472=1067.926,216.491,415.831,173.479,29.549,155.363
C01473=1067.919,216.242,415.857,173.478,29.545,155.362
C01474=1067.914,215.993,415.882,173.475,29.541,155.361
C01475=1067.908,215.745,415.907,173.474,29.537,155.361
C01476=1067.903,215.496,415.933,173.471,29.533,155.360
C01477=1067.897,215.248,415.959,173.469,29.529,155.359
C01478=1067.890,215.000,415.985,173.467,29.525,155.359
C01479=1067.885,214.751,416.011,173.465,29.521,155.358
C01480=1067.878,214.502,416.036,173.463,29.517,155.357
C01481=1067.873,214.253,416.062,173.461,29.513,155.356
C01482=1067.867,214.004,416.087,173.459,29.509,155.356
C01483=1067.861,213.756,416.112,173.457,29.505,155.355
C01484=1067.856,213.507,416.138,173.455,29.501,155.354
C01485=1067.849,213.259,416.164,173.453,29.497,155.354
C01486=1067.843,213.010,416.189,173.451,29.492,155.353
C01487=1067.838,212.761,416.215,173.449,29.489,155.352
C01488=1067.832,212.512,416.240,173.447,29.485,155.352
C01489=1067.826,212.265,416.265,173.445,29.480,155.351
C01490=1067.820,212.016,416.291,173.443,29.476,155.350
C01491=1067.814,211.767,416.316,173.441,29.472,155.350
C01492=1067.808,211.518,416.342,173.439,29.468,155.349
C01493=1067.802,211.270,416.367,173.437,29.464,155.348
C01494=1067.796,211.021,416.392,173.435,29.460,155.348
C01495=1067.791,210.773,416.418,173.433,29.456,155.347
C01496=1067.785,210.524,416.443,173.431,29.452,155.346
C01497=1067.778,210.275,416.469,173.429,29.448,155.346
C01498=1067.772,210.027,416.494,173.427,29.444,155.345
C01499=1067.766,209.778,416.519,173.425,29.440,155.344
C01500=1067.761,209.529,416.544,173.423,29.436,155.343
C01501=1067.755,209.280,416.569,173.421,29.431,155.343
C01502=1067.749,209.064,416.592,173.419,29.428,155.342
C01503=1067.744,208.847,416.614,173.418,29.425,155.341
C01504=1067.740,208.630,416.635,173.416,29.421,155.341
C01505=1067.734,208.414,416.658,173.414,29.417,155.340
C01506=1067.729,208.197,416.679,173.412,29.414,155.340
C01507=1067.724,207.980,416.702,173.410,29.410,155.339
C01508=1067.718,207.763,416.723,173.409,29.407,155.338
C01509=1067.714,207.547,416.745,173.407,29.403,155.338
C01510=1067.689,206.502,416.848,173.259,29.329,155.334
C01511=1067.683,206.253,416.872,173.256,29.325,155.333
C01512=1067.677,206.004,416.896,173.255,29.322,155.333
C01513=1067.672,205.756,416.920,173.252,29.319,155.332
C01514=1067.666,205.507,416.946,173.250,29.316,155.332
C01515=1067.661,205.259,416.970,173.248,29.312,155.331
C01516=1067.655,205.009,416.994,173.245,29.310,155.331
C01517=1067.649,204.761,417.018,173.244,29.306,155.330
C01518=1067.643,204.512,417.042,173.241,29.303,155.330
C01519=1067.637,204.263,417.067,173.239,29.300,155.330
C01520=1067.632,204.015,417.091,173.237,29.297,155.329
C01521=1067.625,203.766,417.115,173.234,29.293,155.329
C01522=1067.620,203.517,417.140,173.233,29.291,155.328
C01523=1067.615,203.268,417.164,173.230,29.287,155.328
C01524=1067.609,203.019,417.188,173.228,29.285,155.327
C01525=1067.604,202.771,417.213,173.226,29.281,155.327
C01526=1067.598,202.522,417.236,173.223,29.278,155.326
C01527=1067.592,202.273,417.261,173.222,29.275,155.326
C01528=1067.586,202.024,417.285,173.219,29.272,155.325
C01529=1067.580,201.776,417.309,173.217,29.269,155.325
C01530=1067.574,201.527,417.334,173.215,29.265,155.324
C01531=1067.568,201.279,417.357,173.212,29.262,155.324
C01532=1067.563,201.029,417.382,173.211,29.259,155.323
C01533=1067.557,200.781,417.405,173.208,29.256,155.323
C01534=1067.552,200.532,417.429,173.206,29.253,155.322
C01535=1067.545,200.283,417.453,173.204,29.250,155.322
C01536=1067.540,200.034,417.477,173.202,29.248,155.322
C01537=1067.534,199.786,417.501,173.200,29.244,155.321
C01538=1067.528,199.537,417.526,173.197,29.241,155.321
C01539=1067.522,199.288,417.549,173.195,29.238,155.320
C01540=1067.517,199.039,417.573,173.193,29.235,155.320
C01541=1067.510,198.790,417.597,173.191,29.232,155.319
C01542=1067.504,198.542,417.620,173.188,29.229,155.319
C01543=1067.499,198.293,417.645,173.187,29.226,155.318
C01544=1067.492,198.044,417.669,173.184,29.223,155.318
C01545=1067.487,197.795,417.692,173.183,29.220,155.317
C01546=1067.481,197.547,417.716,173.180,29.217,155.317
C01547=1067.475,197.298,417.741,173.177,29.214,155.317
C01548=1067.469,197.049,417.764,173.176,29.210,155.316
C01549=1067.464,196.800,417.788,173.173,29.208,155.316
C01550=1067.457,196.551,417.812,173.172,29.204,155.315
C01551=1067.452,196.303,417.836,173.169,29.201,155.315
C01552=1067.446,196.054,417.859,173.167,29.198,155.314
C01553=1067.440,195.805,417.883,173.165,29.195,155.314
C01554=1067.434,195.556,417.907,173.163,29.192,155.313
C01555=1067.429,195.307,417.930,173.161,29.189,155.313
C01556=1067.423,195.059,417.954,173.159,29.186,155.313
C01557=1067.418,194.810,417.977,173.156,29.183,155.312
C01558=1067.412,194.561,418.002,173.155,29.180,155.312
C01559=1067.406,194.312,418.026,173.152,29.177,155.311
C01560=1067.400,194.063,418.049,173.150,29.174,155.311
C01561=1067.395,193.815,418.073,173.148,29.171,155.310
C01562=1067.389,193.566,418.096,173.146,29.168,155.310
C01563=1067.383,193.316,418.120,173.144,29.165,155.309
C01564=1067.377,193.068,418.143,173.142,29.162,155.309
C01565=1067.371,192.819,418.167,173.139,29.159,155.308
C01566=1067.366,192.571,418.191,173.138,29.156,155.308
C01567=1067.360,192.322,418.214,173.135,29.153,155.308
C01568=1067.355,192.073,418.239,173.134,29.150,155.307
C01569=1067.349,191.824,418.262,173.131,29.147,155.307
C01570=1067.343,191.575,418.285,173.129,29.143,155.306
C01571=1067.337,191.293,418.312,173.127,29.140,155.306
C01572=1067.330,191.010,418.339,173.124,29.136,155.305
C01573=1067.324,190.728,418.365,173.122,29.133,155.305
C01574=1067.317,190.445,418.393,173.119,29.129,155.304
C01575=1067.312,190.196,418.416,173.118,29.127,155.304
C01576=1067.306,189.948,418.439,173.115,29.123,155.303
C01577=1067.301,189.698,418.463,173.113,29.121,155.303
C01578=1067.295,189.450,418.486,173.111,29.117,155.302
C01579=1067.289,189.201,418.509,173.109,29.114,155.302
C01580=1067.284,188.952,418.533,173.108,29.112,155.301
C01581=1067.278,188.704,418.557,173.105,29.108,155.301
C01582=1067.272,188.455,418.580,173.103,29.106,155.300
C01583=1067.267,188.206,418.603,173.101,29.102,155.300
C01584=1067.261,187.957,418.627,173.099,29.099,155.300
C01585=1067.255,187.709,418.650,173.097,29.096,155.299
C01586=1067.250,187.459,418.673,173.095,29.093,155.299
C01587=1067.244,187.210,418.697,173.092,29.090,155.298
C01588=1067.238,186.961,418.720,173.091,29.087,155.298
C01589=1067.233,186.712,418.744,173.088,29.084,155.297
C01590=1067.227,186.463,418.767,173.087,29.081,155.297
C01591=1067.221,186.215,418.790,173.085,29.078,155.296
C01592=1067.216,185.966,418.814,173.082,29.075,155.296
C01593=1067.211,185.717,418.837,173.081,29.072,155.295
C01594=1067.205,185.468,418.860,173.078,29.069,155.295
C01595=1067.199,185.219,418.884,173.077,29.066,155.295
C01596=1067.194,184.971,418.907,173.074,29.062,155.294
C01597=1067.188,184.722,418.930,173.072,29.060,155.294
C01598=1067.182,184.473,418.953,173.071,29.057,155.293
C01599=1067.177,184.224,418.976,173.068,29.054,155.293
C01600=1067.171,183.975,418.999,173.067,29.051,155.292
C01601=1067.165,183.726,419.022,173.064,29.048,155.292
C01602=1067.159,183.477,419.045,173.062,29.045,155.291
C01603=1067.153,183.229,419.068,173.060,29.042,155.291
C01604=1067.147,182.980,419.091,173.058,29.040,155.291
C01605=1067.141,182.731,419.114,173.056,29.037,155.290
C01606=1067.135,182.482,419.137,173.054,29.034,155.290
C01607=1067.129,182.233,419.160,173.052,29.031,155.289
C01608=1067.123,181.984,419.183,173.050,29.028,155.289
C01609=1067.118,181.735,419.206,173.048,29.025,155.289
C01610=1067.111,181.487,419.228,173.045,29.022,155.288
C01611=1067.105,181.238,419.251,173.044,29.019,155.288
C01612=1067.100,180.989,419.274,173.042,29.017,155.287
C01613=1067.094,180.740,419.297,173.040,29.013,155.287
C01614=1067.088,180.491,419.320,173.038,29.011,155.286
C01615=1067.082,180.242,419.343,173.035,29.008,155.286
C01616=1067.076,179.993,419.365,173.034,29.005,155.286
C01617=1067.070,179.745,419.388,173.032,29.002,155.285
C01618=1067.065,179.496,419.411,173.030,28.999,155.285
C01619=1067.059,179.247,419.434,173.028,28.996,155.284
C01620=1067.053,178.998,419.457,173.025,28.993,155.284
C01621=1067.048,178.748,419.479,173.024,28.990,155.284
C01622=1067.041,178.500,419.502,173.022,28.988,155.283
C01623=1067.035,178.251,419.524,173.019,28.985,155.283
C01624=1067.030,178.002,419.547,173.018,28.982,155.282
C01625=1067.024,177.753,419.570,173.016,28.979,155.282
C01626=1067.018,177.504,419.593,173.014,28.976,155.281
C01627=1067.012,177.256,419.616,173.012,28.973,155.281
C01628=1067.006,177.006,419.638,173.009,28.970,155.281
C01629=1067.001,176.757,419.661,173.008,28.968,155.280
C01630=1066.995,176.508,419.684,173.006,28.964,155.280
C01631=1066.989,176.259,419.707,173.004,28.961,155.279
C01632=1066.983,176.011,419.729,173.002,28.959,155.279
C01633=1066.977,175.761,419.751,173.000,28.956,155.278
C01634=1066.972,175.512,419.774,172.998,28.953,155.278
C01635=1066.966,175.230,419.800,172.995,28.950,155.278
C01636=1066.958,174.947,419.825,172.994,28.946,155.277
C01637=1066.952,174.664,419.851,172.991,28.943,155.277
C01638=1066.946,174.382,419.877,172.989,28.940,155.276
C01639=1066.940,174.133,419.900,172.987,28.937,155.276
C01640=1066.934,173.884,419.922,172.985,28.934,155.275
C01641=1066.928,173.635,419.945,172.983,28.931,155.275
C01642=1066.922,173.386,419.968,172.981,28.928,155.274
C01643=1066.917,173.136,419.990,172.979,28.926,155.274
C01644=1066.911,172.888,420.012,172.977,28.922,155.273
C01645=1066.905,172.640,420.035,172.975,28.919,155.273
C01646=1066.900,172.390,420.057,172.974,28.917,155.273
C01647=1066.893,172.141,420.079,172.971,28.914,155.272
C01648=1066.888,171.893,420.102,172.969,28.911,155.272
C01649=1066.882,171.643,420.124,172.968,28.908,155.271
C01650=1066.877,171.395,420.147,172.965,28.905,155.271
C01651=1066.871,171.146,420.169,172.964,28.902,155.271
C01652=1066.865,170.897,420.192,172.962,28.899,155.270
C01653=1066.859,170.648,420.215,172.959,28.896,155.270
C01654=1066.853,170.399,420.236,172.958,28.893,155.269
C01655=1066.848,170.150,420.259,172.956,28.890,155.269
C01656=1066.843,169.901,420.281,172.954,28.887,155.268
C01657=1066.837,169.652,420.304,172.952,28.885,155.268
C01658=1066.831,169.403,420.326,172.950,28.882,155.268
C01659=1066.825,169.154,420.349,172.949,28.879,155.267
C01660=1066.820,168.905,420.370,172.946,28.876,155.267
C01661=1066.814,168.656,420.393,172.945,28.873,155.266
C01662=1066.808,168.407,420.415,172.943,28.870,155.266
C01663=1066.803,168.158,420.438,172.941,28.867,155.265
C01664=1066.797,167.910,420.459,172.939,28.864,155.265
C01665=1066.791,167.661,420.482,172.937,28.861,155.265
C01666=1066.786,167.411,420.504,172.935,28.859,155.264
C01667=1066.780,167.163,420.526,172.933,28.856,155.264
C01668=1066.775,166.914,420.549,172.931,28.853,155.263
C01669=1066.769,166.664,420.571,172.930,28.850,155.263
C01670=1066.763,166.416,420.593,172.927,28.847,155.262
C01671=1066.758,166.167,420.615,172.926,28.844,155.262
C01672=1066.752,165.918,420.638,172.924,28.841,155.261
C01673=1066.746,165.669,420.660,172.922,28.838,155.261
C01674=1066.741,165.420,420.681,172.920,28.835,155.261
C01675=1066.735,165.171,420.704,172.918,28.833,155.260
C01676=1066.729,164.922,420.726,172.917,28.830,155.260
C01677=1066.724,164.674,420.749,172.914,28.826,155.259
C01678=1066.719,164.424,420.771,172.913,28.824,155.259
C01679=1066.713,164.175,420.792,172.911,28.821,155.259
C01680=1066.708,163.926,420.814,172.909,28.818,155.258
C01681=1066.702,163.677,420.837,172.907,28.815,155.258
C01682=1066.696,163.428,420.859,172.905,28.812,155.257
C01683=1066.691,163.179,420.881,172.904,28.809,155.257
C01684=1066.685,162.931,420.903,172.902,28.806,155.256
C01685=1066.680,162.682,420.925,172.899,28.803,155.256
C01686=1066.674,162.432,420.947,172.898,28.800,155.255
C01687=1066.668,162.183,420.969,172.896,28.798,155.255
C01688=1066.663,161.935,420.991,172.895,28.795,155.255
C01689=1066.657,161.686,421.013,172.892,28.791,155.254
C01690=1066.652,161.437,421.035,172.890,28.789,155.254
C01691=1066.647,161.187,421.057,172.889,28.786,155.253
C01692=1066.640,160.939,421.080,172.887,28.783,155.253
C01693=1066.635,160.690,421.101,172.885,28.780,155.253
C01694=1066.629,160.441,421.123,172.883,28.777,155.252
C01695=1066.623,160.191,421.145,172.881,28.775,155.252
C01696=1066.617,159.943,421.166,172.880,28.771,155.251
C01697=1066.611,159.694,421.188,172.877,28.769,155.251
C01698=1066.606,159.444,421.210,172.876,28.766,155.250
C01699=1066.599,159.162,421.234,172.873,28.763,155.250
C01700=1066.592,158.878,421.259,172.871,28.760,155.250
C01701=1066.586,158.594,421.284,172.869,28.756,155.249
C01702=1066.580,158.312,421.309,172.867,28.753,155.249
C01703=1066.574,158.062,421.330,172.866,28.751,155.248
C01704=1066.568,157.814,421.351,172.863,28.748,155.248
C01705=1066.563,157.564,421.374,172.862,28.745,155.247
C01706=1066.556,157.315,421.395,172.860,28.742,155.247
C01707=1066.551,157.067,421.417,172.858,28.739,155.246
C01708=1066.545,156.818,421.438,172.856,28.736,155.246
C01709=1066.540,156.569,421.460,172.854,28.733,155.246
C01710=1066.534,156.320,421.482,172.853,28.730,155.245
C01711=1066.528,156.070,421.503,172.851,28.728,155.245
C01712=1066.522,155.822,421.525,172.849,28.725,155.244
C01713=1066.517,155.572,421.547,172.847,28.722,155.244
C01714=1066.511,155.324,421.568,172.845,28.719,155.244
C01715=1066.505,155.075,421.590,172.844,28.717,155.243
C01716=1066.499,154.825,421.611,172.842,28.714,155.243
C01717=1066.493,154.577,421.633,172.839,28.711,155.242
C01718=1066.487,154.328,421.654,172.838,28.708,155.242
C01719=1066.482,154.079,421.676,172.836,28.705,155.242
C01720=1066.476,153.830,421.698,172.835,28.702,155.241
C01721=1066.470,153.581,421.719,172.833,28.699,155.241
C01722=1066.464,153.332,421.741,172.830,28.697,155.240
C01723=1066.458,153.082,421.762,172.829,28.694,155.240
C01724=1066.453,152.834,421.783,172.827,28.691,155.240
C01725=1066.447,152.584,421.805,172.826,28.688,155.239
C01726=1066.441,152.336,421.826,172.824,28.686,155.239
C01727=1066.435,152.087,421.847,172.821,28.683,155.238
C01728=1066.430,151.838,421.869,172.820,28.680,155.238
C01729=1066.424,151.588,421.890,172.818,28.677,155.237
C01730=1066.419,151.340,421.911,172.817,28.674,155.237
C01731=1066.413,151.090,421.933,172.815,28.672,155.237
C01732=1066.407,150.842,421.954,172.812,28.669,155.236
C01733=1066.401,150.593,421.976,172.811,28.666,155.236
C01734=1066.396,150.344,421.997,172.809,28.663,155.235
C01735=1066.389,150.094,422.018,172.808,28.661,155.235
C01736=1066.384,149.846,422.039,172.806,28.658,155.235
C01737=1066.378,149.597,422.061,172.804,28.655,155.234
C01738=1066.372,149.347,422.082,172.802,28.652,155.234
C01739=1066.366,149.098,422.103,172.800,28.649,155.233
C01740=1066.361,148.850,422.125,172.799,28.646,155.233
C01741=1066.355,148.600,422.146,172.797,28.643,155.233
C01742=1066.349,148.351,422.167,172.795,28.641,155.232
C01743=1066.343,148.102,422.188,172.794,28.638,155.232
C01744=1066.338,147.853,422.209,172.791,28.635,155.231
C01745=1066.332,147.604,422.231,172.790,28.632,155.231
C01746=1066.326,147.355,422.252,172.788,28.629,155.231
C01747=1066.320,147.106,422.273,172.786,28.627,155.230
C01748=1066.315,146.857,422.294,172.785,28.624,155.230
C01749=1066.309,146.608,422.316,172.782,28.621,155.229
C01750=1066.303,146.359,422.336,172.781,28.618,155.229
C01751=1066.297,146.111,422.357,172.779,28.616,155.229
C01752=1066.291,145.861,422.378,172.777,28.613,155.228
C01753=1066.286,145.612,422.399,172.776,28.610,155.228
C01754=1066.279,145.363,422.421,172.774,28.607,155.227
C01755=1066.274,145.114,422.441,172.773,28.605,155.227
C01756=1066.268,144.865,422.463,172.770,28.602,155.227
C01757=1066.263,144.616,422.483,172.768,28.599,155.226
C01758=1066.256,144.367,422.505,172.767,28.596,155.226
C01759=1066.251,144.118,422.525,172.765,28.593,155.225
C01760=1066.245,143.869,422.546,172.764,28.591,155.225
C01761=1066.239,143.619,422.567,172.762,28.588,155.224
C01762=1066.234,143.371,422.589,172.759,28.585,155.224
C01763=1066.227,143.087,422.613,172.758,28.582,155.224
C01764=1066.220,142.804,422.636,172.756,28.579,155.223
C01765=1066.213,142.520,422.660,172.754,28.575,155.223
C01766=1066.207,142.236,422.683,172.752,28.573,155.222
C01767=1066.202,141.988,422.704,172.751,28.570,155.222
C01768=1066.196,141.738,422.725,172.748,28.567,155.221
C01769=1066.190,141.489,422.747,172.747,28.564,155.221
C01770=1066.184,141.241,422.767,172.745,28.561,155.221
C01771=1066.178,140.991,422.788,172.743,28.559,155.220
C01772=1066.173,140.742,422.809,172.742,28.556,155.220
C01773=1066.167,140.492,422.830,172.740,28.553,155.219
C01774=1066.161,140.244,422.851,172.739,28.550,155.219
C01775=1066.155,139.995,422.871,172.737,28.547,155.219
C01776=1066.150,139.745,422.892,172.734,28.545,155.218
C01777=1066.144,139.497,422.913,172.733,28.542,155.218
C01778=1066.138,139.248,422.933,172.731,28.539,155.217
C01779=1066.132,138.998,422.954,172.730,28.537,155.217
C01780=1066.127,138.750,422.975,172.728,28.534,155.217
C01781=1066.121,138.501,422.995,172.726,28.531,155.216
C01782=1066.115,138.251,423.016,172.725,28.528,155.216
C01783=1066.109,138.002,423.037,172.723,28.526,155.215
C01784=1066.103,137.754,423.057,172.721,28.523,155.215
C01785=1066.097,137.504,423.078,172.719,28.520,155.215
C01786=1066.092,137.255,423.099,172.717,28.517,155.214
C01787=1066.086,137.007,423.120,172.716,28.514,155.214
C01788=1066.080,136.757,423.140,172.714,28.512,155.213
C01789=1066.074,136.508,423.160,172.713,28.509,155.213
C01790=1066.069,136.259,423.181,172.711,28.506,155.213
C01791=1066.063,136.009,423.202,172.709,28.503,155.212
C01792=1066.056,135.761,423.223,172.708,28.501,155.212
C01793=1066.051,135.512,423.243,172.706,28.498,155.211
C01794=1066.045,135.262,423.263,172.704,28.495,155.211
C01795=1066.039,135.013,423.284,172.702,28.492,155.211
C01796=1066.033,134.764,423.304,172.701,28.489,155.210
C01797=1066.028,134.516,423.325,172.699,28.487,155.210
C01798=1066.022,134.266,423.346,172.697,28.484,155.209
C01799=1066.016,134.017,423.366,172.696,28.481,155.209
C01800=1066.011,133.768,423.387,172.694,28.478,155.209
C01801=1066.004,133.518,423.407,172.693,28.476,155.208
C01802=1065.999,133.269,423.428,172.691,28.473,155.208
C01803=1065.993,133.020,423.448,172.689,28.470,155.207
C01804=1065.988,132.771,423.468,172.687,28.467,155.207
C01805=1065.982,132.522,423.489,172.685,28.465,155.207
C01806=1065.975,132.273,423.510,172.684,28.462,155.206
C01807=1065.970,132.024,423.530,172.682,28.459,155.206
C01808=1065.964,131.775,423.550,172.680,28.456,155.205
C01809=1065.958,131.526,423.571,172.679,28.454,155.205
